// TIA Portal project "OCS_Portable_S300_To_S1500" (V14)

(* hardware
DEVICE "S7300/ET200M station_1"  S7-300 station
   slot 0: "Rail_0"  Rail  6ES7 390-1***0-0AA0
   slot 2: "PLC_1"  CPU 317-2 PN/DP  6ES7 317-2EK14-0AB0  V3.2
      slot 2: "PROFINET interface_1"  PN-IO
         slot 1: "Port_1"  Port
         slot 2: "Port_2"  Port
DEVICE "ET 200SP station_1"  ET 200SP-Station
   slot 0: "Rack_0"  Rack  6ES5 710-8MAx1
   slot 1: "PLC_2"  CPU 1512SP-1 PN  6ES7 512-1DK01-0AB0  V2.1
   slot 2: "TM Count 1x24V_1"  TM Count 1x24V  6ES7 138-6AA00-0BA0  V1.2
      slot 1: "TM Count 1x24V_1"  TM Count 1x24V
   slot 3: "CM PtP_1"  CM PtP  6ES7 137-6AA00-0BA0  V1.0
      slot 1: "CM PtP_1"  CM PtP Sub
   slot 4: "TM Pulse 2x24V_1"  TM Pulse 2x24V  6ES7 138-6DB00-0BB1  V1.0
      slot 1: "TM Pulse 2x24V_1"  TM Pulse 2x24V
   slot 5: "Server module_1"  Server module  6ES7 193-6PA00-0AA0  V1.1
      slot 1: "Server module_1"  Server module
   slot 127: "BA 2xRJ45"  BA 2xRJ45  6ES7 193-6AR00-0AA0  V0.0
      slot 32769: "Port_1"  6ES7 193-6AR00-0AA0
      slot 32770: "Port_2"  6ES7 193-6AR00-0AA0
*)

// ===== PLC "PLC_1"  CPU 317-2 PN/DP =====

VAR_GLOBAL   // PLC tag table "Merkers"
   "OSC_Work" AT %M20.5 : Bool;
END_VAR

DATA_BLOCK "Temp"   // DB1
{ S7_Optimized_Access := 'FALSE' }
VERSION : 0.1
   VAR
      Radians : Real;
   END_VAR
BEGIN
END_DATA_BLOCK

DATA_BLOCK "SU"   // DB101
{ S7_Optimized_Access := 'FALSE' }
VERSION : 0.1
   VAR
      su_Uac_6kV : Real;   // Действующее линейное напряжение AC на входе ЯВВ, В
      Spare_4_0 : Int;   // Резерв
      su_Fan_MD_QF1 : Bool;   // Автомат вентиляторов QF1 (0-выкл,1-вкл)
      su_Fan_MD_QF2 : Bool;   // Автомат вентиляторов QF2 (0-выкл,1-вкл)
      su_Fan_MD_QF3 : Bool;   // Автомат вентиляторов QF3 (0-выкл,1-вкл)
      su_Fan_MD_QF4 : Bool;   // Автомат вентиляторов QF4 (0-выкл,1-вкл)
      su_Fan_M1_ON : Bool;   // Контактор вентилятора КМ1 (0-выкл,1-вкл)
      su_Fan_M2_ON : Bool;   // Контактор вентилятора КМ2 (0-выкл,1-вкл)
      su_Fan_M6_ON : Bool;   // Контактор вентилятора КМ6 (0-выкл,1-вкл)
      su_Fan_M7_ON : Bool;   // Контактор вентилятора КМ7 (0-выкл,1-вкл)
      su_Fan_M8_ON : Bool;   // Контактор вентилятора КМ8 (0-выкл,1-вкл)
      su_Temp_ok : Bool;   // Температура в норме (0-выкл,1-вкл)
      su_Fan_MD_Ready : Bool;   // Готовность вентиляции ГП (0-выкл,1-вкл)
      su_Fan_M3_ON : Bool;   // Контактор вентилятора КМ3 (0-выкл,1-вкл)
      su_Fan_M4_ON : Bool;   // Контактор вентилятора КМ4 (0-выкл,1-вкл)
      su_Fan_M5_ON : Bool;   // Контактор вентилятора КМ5 (0-выкл,1-вкл)
      su_LH : Real;   // Длина подъемного каната, м
      su_LC : Real;   // Длина выдвижения рукояти, м
      su_OHRVD_AF : Bool;   // Ограничение хода рукояти. При выдвижении (0-ограничение выкл,1-ограничение)
      su_OHRVT_AF : Bool;   // Ограничение хода рукояти. При втягивании (0-ограничение выкл,1-ограничение)
      su_LC_Reset : Bool;   // Обнулить знчение энкодера напора (1-обнулить)
      su_OPK_AF : Bool;   // Ограничение подъема ковша (0-ограничение выкл, 1-ограничение)
      su_LH_Reset : Bool;   // Обнулить знчение энкодера подъема (1-обнулить)
      su_Field_Reduction : Bool;   // Ослабление поля (0-выкл,1-вкл)
      su_Field_Forcing : Bool;   // Форсировка поля (0-выкл,1-вкл)
      su_Autobrake_ON : Bool;   // Подхват тормозов (0-выкл,1-вкл)
      su_Brake_H : Bool;   // Тормоза привода подъема (1–расторможен,0–заторможен)
      su_Brake_C : Bool;   // Тормоза привода напора (1–расторможен,0–заторможен)
      su_Brake_S : Bool;   // Тормоза привода поворота (1–расторможен,0–заторможен)
      su_Brake_P : Bool;   // Тормоза привода хода левого (1–расторможен,0–заторможен)
      su_Brake_P_R : Bool;   // Тормоза привода хода правого (1–расторможен,0–заторможен)
      su_All_Protect : Bool;   // Автоматические защиты (0-выкл,1–вкл)
      su_BOS_Connect : Bool;   // Связь с БОС (0-связь есть,1-связи нет)
      su_Job_Limit : Bool;   // Уровень ограничения задания (0-задание 100%,1-задание 70%)
      su_Blocking_1 : Bool;   // Блокировка 1 Защита выше напорного вала (1-вкл,0-выкл)
      su_Blocking_2 : Bool;   // Блокировка 2 Защита при збросе ковша (1-вкл,0-выкл)
      su_Blocking_3 : Bool;   // Блокировка 3 Ограничение хода рукояти (1-вкл,0-выкл)
      su_Blocking_4 : Bool;   // Блокировка 4 Ограничение подъема ковша (1-вкл,0-выкл)
      su_Blocking_5 : Bool;   // Блокировка 5 Ограничение боковых нагрузок при черпании(1-вкл,0-выкл)
      su_Blocking_6 : Bool;   // Блокировка 6 Ограничение боковых нагрузок при работе с негабаритами(1-вкл,0-вык
      su_Blocking_7 : Bool;   // Блокировка 7 Передняя кромка(1-вкл,0-выкл)
      su_Blocking_8 : Bool;   // Блокировка 8 Защита от заброса стрелы(1-вкл,0-выкл)
      su_Blocking_9 : Bool;   // Блокировка 9 Ограничение длины разматывания подъемного каната (1-вкл,0-выкл)
      su_Enc_C_Connect : Bool;   // Энкодер напора подключен (1-связь есть,0-связи нет)
      su_Enc_H_Connect : Bool;   // Энкодер подъема подключен (1-связь есть,0-связи нет)
      Spare_19_3 : Bool;   // Резерв
      Spare_19_4 : Bool;   // Резерв
      Spare_19_5 : Bool;   // Резерв
      Spare_19_6 : Bool;   // Резерв
      Spare_19_7 : Bool;   // Резерв
      su_Job_H : DInt := DINT#0;   // Задание для привода подъема
      su_Job_S : DInt := DINT#0;   // Задание для привода поворота
      Spare_28_0 : Int;   // Резерв
      su_Excav : Bool;   // Режим "Экскавация" (1-вкл,0-выкл)
      su_Prop : Bool;   // Режим "Ход" (1-вкл,0-выкл)
      su_Work_S : Bool;   // Привод поворота расторможен (1-вкл,0-выкл)
      su_Work_C : Bool;   // Привод напора расторможен (1-вкл,0-выкл)
      su_Work_H : Bool;   // Привод подъема расторможен (1-вкл,0-выкл)
      su_Ready_S : Bool;   // Разрешение растормозить привод поворота (1-вкл,0-выкл)
      su_Fan_Prop : Bool;   // Вентиляторы двигателей хода (1-вкл,0-выкл)
      su_AR_Mode_Work : Bool;   // Активные выпрямители в режиме "Работа" (1-вкл,0-выкл)
      su_Ctrl_Is : Bool;   // Контроль изоляции (1-вкл,0-выкл)
      su_Ctrl_Ladder : Bool;   // Контроль положения лестницы (1-вкл,0-выкл)
      su_Relay_Alarm_ON : Bool;   // Реле включения аварии (1-вкл,0-выкл)
      su_Relay_CtrlC : Bool;   // Реле включения цепей управления (1-вкл,0-выкл)
      su_Ctrl_Breaker : Bool;   // Контроль состояния вводных автоматов (1-вкл,0-выкл)
      su_Limit_Switch : Bool;   // Конечные выключатели шкафов управления (1-вкл,0-выкл)
      su_Ready_P : Bool;   // Разрешение растормозить привод хода (1-вкл,0-выкл)
      su_Fan_Mot : Bool;   // Вентиляция машин (1-вкл,0-выкл)
      su_Work_P : Bool;   // Привод хода расторможен (1-вкл,0-выкл)
      su_Lubr : Bool;   // Смазка редукторов поворота (1-вкл,0-выкл)
      su_BUP_StartUp_ARm : Bool;   // Блок управления в режиме инициализации (1-вкл,0-выкл)
      su_BUP_ON_ARm : Bool;   // Блок управления в работе, управляющие импульсы поданы (1-вкл,0-выкл)
      su_BUP_StartUp_ARs1 : Bool;   // Блок управления в режиме инициализации (1-вкл,0-выкл)
      su_BUP_ON_ARs1 : Bool;   // Блок управления в работе, управляющие импульсы поданы (1-вкл,0-выкл)
      su_BUP_StartUp_ARs2 : Bool;   // Блок управления в режиме инициализации (1-вкл,0-выкл)
      su_BUP_ON_ARs2 : Bool;   // Блок управления в работе, управляющие импульсы поданы (1-вкл,0-выкл)
      su_BUP_StartUp_ARs3 : Bool;   // Блок управления в режиме инициализации (1-вкл,0-выкл)
      su_BUP_ON_ARs3 : Bool;   // Блок управления в работе, управляющие импульсы поданы (1-вкл,0-выкл)
      su_Magnet_M1H : Bool;   // Двигатель намагничен (1-вкл,0-выкл)
      su_BUP_StartUp_Hm : Bool;   // Блок управления в режиме инициализации (1-вкл,0-выкл)
      su_BUP_ON_Hm : Bool;   // Блок управления в работе, управляющие импульсы поданы (1-вкл,0-выкл)
      su_Magnet_M2H : Bool;   // Двигатель намагничен (1-вкл,0-выкл)
      su_BUP_StartUp_Hs : Bool;   // Блок управления в режиме инициализации (1-вкл,0-выкл)
      su_BUP_ON_Hs : Bool;   // Блок управления в работе, управляющие импульсы поданы (1-вкл,0-выкл)
      su_Magnet_MC : Bool;   // Двигатель намагничен (1-вкл,0-выкл)
      su_BUP_StartUp_C : Bool;   // Блок управления в режиме инициализации (1-вкл,0-выкл)
      su_BUP_ON_C : Bool;   // Блок управления в работе, управляющие импульсы поданы (1-вкл,0-выкл)
      su_Magnet_M1S : Bool;   // Двигатель намагничен (1-вкл,0-выкл)
      su_BUP_StartUp_Sm : Bool;   // Блок управления в режиме инициализации (1-вкл,0-выкл)
      su_BUP_ON_Sm : Bool;   // Блок управления в работе, управляющие импульсы поданы (1-вкл,0-выкл)
      su_Magnet_M2S : Bool;   // Двигатель намагничен (1-вкл,0-выкл)
      su_BUP_StartUp_Ss1 : Bool;   // Блок управления в режиме инициализации (1-вкл,0-выкл)
      su_BUP_ON_Ss1 : Bool;   // Блок управления в работе, управляющие импульсы поданы (1-вкл,0-выкл)
      su_Magnet_M3S : Bool;   // Двигатель намагничен (1-вкл,0-выкл)
      su_BUP_StartUp_Ss2 : Bool;   // Блок управления в режиме инициализации (1-вкл,0-выкл)
      su_BUP_ON_Ss2 : Bool;   // Блок управления в работе, управляющие импульсы поданы (1-вкл,0-выкл)
      su_Magnet_M4S : Bool;   // Двигатель намагничен (1-вкл,0-выкл)
      su_BUP_StartUp_Ss3 : Bool;   // Блок управления в режиме инициализации (1-вкл,0-выкл)
      su_BUP_ON_Ss3 : Bool;   // Блок управления в работе, управляющие импульсы поданы (1-вкл,0-выкл)
      su_Magnet_M1P : Bool;   // Двигатель намагничен (1-вкл,0-выкл)
      su_BUP_StartUp_C_P : Bool;   // Блок управления в режиме инициализации (1-вкл,0-выкл)
      su_BUP_ON_C_P : Bool;   // Блок управления в работе, управляющие импульсы поданы (1-вкл,0-выкл)
      su_Magnet_M2P : Bool;   // Двигатель намагничен (1-вкл,0-выкл)
      su_BUP_StartUp_S_P : Bool;   // Блок управления в режиме инициализации (1-вкл,0-выкл)
      su_BUP_ON_S_P : Bool;   // Блок управления в работе, управляющие импульсы поданы (1-вкл,0-выкл)
      Spare_36_5 : Bool;   // Резерв
      Spare_36_6 : Bool;   // Резерв
      Spare_36_7 : Bool;   // Резерв
      Spare_37_B : Byte;   // Резерв
      su_I_ARm : Real;   // Действующий ток, А
      su_Ud_ARm : Real;   // Напряжение звена постоянного тока, В
      su_Ia_ARm : Real;   // Амплитудный активный ток выпрямителя, А
      su_Ir_ARm : Real;   // Амплитудный индуктивный ток выпрямителя, А
      su_fs_ARm : Real;   // Частота сети
      su_Us_ARm : Real;   // Амплитудное напряжение на входе выпрямителя
      su_Pa_ARm : Real;   // Активная мощность выпрямителя
      su_I_ARs1 : Real;   // Действующий ток, А
      su_Ud_ARs1 : Real;   // Напряжение звена постоянного тока, В
      su_Ia_ARs1 : Real;   // Амплитудный активный ток выпрямителя, А
      su_Ir_ARs1 : Real;   // Амплитудный индуктивный ток выпрямителя, А
      su_fs_ARs1 : Real;   // Частота сети
      su_Us_ARs1 : Real;   // Амплитудное напряжение на входе выпрямителя
      su_Pa_ARs1 : Real;   // Активная мощность выпрямителя
      su_Job_I_ARs1 : Real;   // Задание на регулятор тока ведомого выпрямителя
      su_I_ARs2 : Real;   // Действующий ток, А
      su_Ud_ARs2 : Real;   // Напряжение звена постоянного тока, В
      su_Ia_ARs2 : Real;   // Амплитудный активный ток выпрямителя, А
      su_Ir_ARs2 : Real;   // Амплитудный индуктивный ток выпрямителя, А
      su_fs_ARs2 : Real;   // Частота сети
      su_Us_ARs2 : Real;   // Амплитудное напряжение на входе выпрямителя
      su_Pa_ARs2 : Real;   // Активная мощность выпрямителя
      su_Job_I_ARs2 : Real;   // Задание на регулятор тока ведомого выпрямителя
      su_I_ARs3 : Real;   // Действующий ток, А
      su_Ud_ARs3 : Real;   // Напряжение звена постоянного тока, В
      su_Ia_ARs3 : Real;   // Амплитудный активный ток выпрямителя, А
      su_Ir_ARs3 : Real;   // Амплитудный индуктивный ток выпрямителя, А
      su_fs_ARs3 : Real;   // Частота сети
      su_Us_ARs3 : Real;   // Амплитудное напряжение на входе выпрямителя
      su_Pa_ARs3 : Real;   // Активная мощность выпрямителя
      su_Job_I_ARs3 : Real;   // Задание на регулятор тока ведомого выпрямителя
      su_I_M1H : Real;   // Действующий ток статора, А
      su_Ud_Hm : Real;   // Напряжение звена постоянного тока, В
      su_Id_M1H : Real;   // Ток намагничивания статора, А
      su_Iq_M1H : Real;   // Активный ток статора, А
      su_W_M1H : Real;   // Скорость, рад/с
      su_Psi2_M1H : Real;   // Поток ротора, Вб
      su_U_M1H : Real;   // Фазное напряжение двигателя, В
      su_JobW_Hm : Real;   // Задание на скорость, ед
      su_I_M2H : Real;   // Действующий ток статора, А
      su_Ud_Hs : Real;   // Напряжение звена постоянного тока, В
      su_Id_M2H : Real;   // Ток намагничивания статора, А
      su_Iq_M2H : Real;   // Активный ток статора, А
      su_W_M2H : Real;   // Скорость, рад/с
      su_Psi2_M2H : Real;   // Поток ротора, Вб
      su_U_M2H : Real;   // Фазное напряжение двигателя, В
      su_JobW_Hs : Real;   // Задание на скорость, ед
      su_I_MC : Real;   // Действующий ток статора, А
      su_Ud_C : Real;   // Напряжение звена постоянного тока, В
      su_Id_MC : Real;   // Ток намагничивания статора, А
      su_Iq_MC : Real;   // Активный ток статора, А
      su_W_MC : Real;   // Скорость, рад/с
      su_Psi2_MC : Real;   // Поток ротора, Вб
      su_U_MC : Real;   // Фазное напряжение двигателя, В
      su_JobW_C : Real;   // Задание на скорость, ед
      su_I_M1S : Real;   // Действующий ток статора, А
      su_Ud_Sm : Real;   // Напряжение звена постоянного тока, В
      su_Id_M1S : Real;   // Ток намагничивания статора, А
      su_Iq_M1S : Real;   // Активный ток статора, А
      su_W_M1S : Real;   // Скорость, рад/с
      su_Psi2_M1S : Real;   // Поток ротора, Вб
      su_U_M1S : Real;   // Фазное напряжение двигателя, В
      su_JobW_Sm : Real;   // Задание на скорость, ед
      su_I_M2S : Real;   // Действующий ток статора, А
      su_Ud_Ss1 : Real;   // Напряжение звена постоянного тока, В
      su_Id_M2S : Real;   // Ток намагничивания статора, А
      su_Iq_M2S : Real;   // Активный ток статора, А
      su_W_M2S : Real;   // Скорость, рад/с
      su_Psi2_M2S : Real;   // Поток ротора, Вб
      su_U_M2S : Real;   // Фазное напряжение двигателя, В
      su_JobW_Ss1 : Real;   // Задание на скорость, ед
      Spare_322_0 : Real;   // Резерв
      su_State_H1 : Bool;   // Готовность преобразователя подъема 1 (0-авария,1-готов)
      su_State_H2 : Bool;   // Готовность преобразователя подъема 2 (0-авария,1-готов)
      su_State_C : Bool;   // Готовность преобразователя напора (0-авария,1-готов)
      su_State_P1 : Bool;   // Готовность преобразователя хода 1 (0-авария,1-готов)
      su_State_P2 : Bool;   // Готовность преобразователя хода 2 (0-авария,1-готов)
      su_State_S1 : Bool;   // Готовность преобразователя поворота 1 (0-авария,1-готов)
      su_Overheat_TS : Bool;   // Перегрев силового трансформатора (0-авария,1-готов)
      su_GB_Charge : Bool;   // Блок заряда аккумуляторов (0-авария,1-готов)
      su_Relay_K4 : Bool;   // Реле К4 резерв (0-выкл,1-вкл)
      su_Relay_K3 : Bool;   // Реле К3, готовность блоков сброса (0-выкл,1-вкл)
      su_Relay_K2 : Bool;   // Реле К2 включение ВВ контактора (0-выкл,1-вкл)
      su_State_AR1 : Bool;   // Готовность активного выпрямителя 1 (0-авария,1-готов)
      su_State_AR2 : Bool;   // Готовность активного выпрямителя 2 (0-авария,1-готов)
      su_State_AR3 : Bool;   // Готовность активного выпрямителя 3 (0-авария,1-готов)
      su_State_Chop1 : Bool;   // Блок сброс 1 (0-авария,1-готов)
      su_State_Chop2 : Bool;   // Блок сброс 2 (0-авария,1-готов)
      su_Relay_K7 : Bool;   // Реле К7 резерв (0-выкл,1-вкл)
      su_Relay_K6 : Bool;   // Реле К6 резерв (0-выкл,1-вкл)
      su_State_AR4 : Bool;   // Готовность активного выпрямителя 4 (0-авария,1-готов)
      su_Relay_K5 : Bool;   // Реле К5 резерв (0-выкл,1-вкл)
      su_Relay_K1 : Bool;   // Реле К1 включение готовности преобразователей ГП (0-выкл,1-вкл)
      su_Vent_MD : Bool;   // Вентиляция главных приводов (0-выкл,1-вкл)
      su_HV_Contactor_ON : Bool;   // ВВ контактор включен (0-выкл,1-вкл)
      su_State_S2 : Bool;   // Готовность преобразователя поворота 2 (0-авария,1-готов)
      su_State_S3 : Bool;   // Готовность преобразователя поворота 3 (0-авария,1-готов)
      su_State_S4 : Bool;   // Готовность преобразователя поворота 4 (0-авария,1-готов)
      Spare_329_2 : Bool;   // Резерв
      Spare_329_3 : Bool;   // Резерв
      Spare_329_4 : Bool;   // Резерв
      Spare_329_5 : Bool;   // Резерв
      Spare_329_6 : Bool;   // Резерв
      Spare_329_7 : Bool;   // Резерв
      su_BOS_Enc_H : Int;   // Значение БОСЭ механизма подъема (1 оборот 2^10 бит)
      su_BOS_Enc_C : Int;   // Значение БОСЭ механизма напора (1 оборот 2^10 бит)
      su_MD_OFF : Bool;   // Отключение главных приводов (0-выкл,1-вкл)
      su_VH : Real;   // Линейная скорость подъема
      su_VC : Real;   // Линейная скорость напора
      su_Job_C : DInt := DINT#0;   // Задание для привода напора
      su_Ia_PowerT : Real;   // Ток в фазе А первичной обмотки силового трансформатора, А
      su_Ib_PowerT : Real;   // Ток в фазе В первичной обмотки силового трансформатора, А
      su_I_M3S : Real;   // Действующий ток статора, А
      su_Ud_Ss2 : Real;   // Напряжение звена постоянного тока, В
      su_Id_M3S : Real;   // Ток намагничивания статора, А
      su_Iq_M3S : Real;   // Активный ток статора, А
      su_W_M3S : Real;   // Скорость, рад/с
      su_Psi2_M3S : Real;   // Поток ротора, Вб
      su_U_M3S : Real;   // Фазное напряжение двигателя, В
      su_JobW_Ss2 : Real;   // Задание на скорость, ед
      su_I_M4S : Real;   // Действующий ток статора, А
      su_Ud_Ss3 : Real;   // Напряжение звена постоянного тока, В
      su_Id_M4S : Real;   // Ток намагничивания статора, А
      su_Iq_M4S : Real;   // Активный ток статора, А
      su_W_M4S : Real;   // Скорость, рад/с
      su_Psi2_M4S : Real;   // Поток ротора, Вб
      su_U_M4S : Real;   // Фазное напряжение двигателя, В
      su_JobW_Ss3 : Real;   // Задание на скорость, ед
      su_I_M1P : Real;   // Действующий ток статора, А
      su_Ud_C_P : Real;   // Напряжение звена постоянного тока, В
      su_Id_M1P : Real;   // Ток намагничивания статора, А
      su_Iq_M1P : Real;   // Активный ток статора, А
      su_W_M1P : Real;   // Скорость, рад/с
      su_Psi2_M1P : Real;   // Поток ротора, Вб
      su_U_M1P : Real;   // Фазное напряжение двигателя, В
      su_JobW_C_P : Real;   // Задание на скорость, ед
      su_I_M2P : Real;   // Действующий ток статора, А
      su_Ud_S_P : Real;   // Напряжение звена постоянного тока, В
      su_Id_M2P : Real;   // Ток намагничивания статора, А
      su_Iq_M2P : Real;   // Активный ток статора, А
      su_W_M2P : Real;   // Скорость, рад/с
      su_Psi2_M2P : Real;   // Поток ротора, Вб
      su_U_M2P : Real;   // Фазное напряжение двигателя, В
      su_JobW_S_P : Real;   // Задание на скорость, ед
      su_BUARm_ID : Int;   // Номер блока активного выпрямителя ведущего
      su_BUARs1_ID : Int;   // Номер блока активного выпрямителя ведомого 1
      su_BUARs2_ID : Int;   // Номер блока активного выпрямителя ведомого 2
      su_BUARs3_ID : Int;   // Номер блока активного выпрямителя ведомого 3
      su_Type_AR : Int;   // Текущий тип преобразователя
      su_BUP_Hm_ID : Int;   // Номер БУПа привода подъема ведущего
      su_BUP_Hs_ID : Int;   // Номер БУПа привода подъема ведомого
      su_BUP_C_ID : Int;   // Номер БУПа привода напора
      su_BUP_Sm_ID : Int;   // Номер БУПа привода поворота ведущего
      su_BUP_Ss1_ID : Int;   // Номер БУПа привода поворота ведомого 1
      su_BUP_Ss2_ID : Int;   // Номер БУПа привода поворота ведомого 2
      su_BUP_Ss3_ID : Int;   // Номер БУПа привода поворота ведомого 3
      su_BUP_CP_ID : Int;   // Номер БУПа привода напора-хода
      su_BUP_SP_ID : Int;   // Номер БУПа привода поворота-хода
      su_Type_Pr : Int;   // Текущий тип привода
      su_Temp_ARm : Int;   // Средняя температура активного выпрямителя ведущего
      su_Temp_ARs1 : Int;   // Средняя температура активного выпрямителя ведомого 1
      su_Temp_ARs3 : Int;   // Средняя температура активного выпрямителя ведомого 2
      su_Temp_ARs2 : Int;   // Средняя температура активного выпрямителя ведомого 3
      su_Temp_Hm : Int;   // Средняя температура преобразователя подъема ведущего
      su_Wr_M1H : Int;   // Электрическая скорость ротора M1H (показания датчика, рад/с)
      su_Temp_Hs : Int;   // Средняя температура преобразователя подъема ведомого
      su_Wr_M2H : Int;   // Электрическая скорость ротора M2H (показания датчика, рад/с)
      su_Temp_C : Int;   // Средняя температура преобразователя напора
      su_Wr_MC : Int;   // Электрическая скорость ротора MC (показания датчика, рад/с)
      su_Temp_Sm : Int;   // Средняя температура преобразователя поворота ведущего
      su_Wr_M1S : Int;   // Электрическая скорость ротора M1S (показания датчика, рад/с)
      su_Temp_Ss1 : Int;   // Средняя температура преобразователя поворота ведомого 1
      su_Wr_M2S : Int;   // Электрическая скорость ротора M2S (показания датчика, рад/с)
      su_Temp_Ss2 : Int;   // Средняя температура преобразователя поворота ведомого 2
      su_Wr_M3S : Int;   // Электрическая скорость ротора M3S (показания датчика, рад/с)
      su_Temp_Ss3 : Int;   // Средняя температура преобразователя поворота ведомого 3
      su_Wr_M4S : Int;   // Электрическая скорость ротора M4S (показания датчика, рад/с)
      su_Temp_C_P : Int;   // Средняя температура преобразователя напора-хода
      su_Wr_M1P : Int;   // Электрическая скорость ротора M1P (показания датчика, рад/с)
      su_Temp_S_P : Int;   // Средняя температура преобразователя поворота-хода
      su_Wr_M2P : Int;   // Электрическая скорость ротора M2P (показания датчика, рад/с)
      su_I_M1H_fs : Real;   // Действующий ток статора, A (быстрое значение)
      su_Id_M1H_fs : Real;   // Ток намагничивания статора, А (быстрое значение)
      su_Iq_M1H_fs : Real := -0.375;   // Активный ток статора, А (быстрое значение)
      su_W_M1H_fs : Real;   // Скорость, рад/с (быстрое значение)
      su_I_C_fs : Real;   // Действующий ток статора, A (быстрое значение)
      su_Id_C_fs : Real;   // Ток намагничивания статора, А (быстрое значение)
      su_Iq_C_fs : Real;   // Активный ток статора, А (быстрое значение)
      su_W_C_fs : Real;   // Скорость, рад/с (быстрое значение)
      su_I_S_fs : Real;   // Действующий ток статора, A (быстрое значение)
      su_Id_S_fs : Real;   // Ток намагничивания статора, А (быстрое значение)
      su_Iq_S_fs : Real := 59.75;   // Активный ток статора, А (быстрое значение)
      su_W_S_fs : Real;   // Скорость, рад/с (быстрое значение)
   END_VAR
BEGIN
END_DATA_BLOCK

DATA_BLOCK "AP"   // DB103
{ S7_Optimized_Access := 'FALSE' }
VERSION : 0.1
   VAR
      ap_QF_FanMD_Off : Bool;   // отключен автомат вентиляторов главных приводов
      ap_UZ_FanMD_On : Bool;   // преобразователь пуска вентиляторов главных приводов включен
      ap_QF_FanProp_Off : Bool;   // отключен автомат вентиляторов двигателей хода
      ap_UZ_FanProp_On : Bool;   // преобразователь пуска вентиляторов двигателей хода включен
      ap_QF_KB_On : Bool;   // автомат преобразователя кабельного барабана включен
      ap_QF_ODK_On : Bool;   // автомат преобразователя открывания днища ковша включен
      ap_PS_110v_On : Bool;   // питание источника 110В включено
      ap_CtrlC_110v_On : Bool;   // питание цепей управления 110В включено
      ap_Gudok : Bool;   // пневмосигнал включен
      ap_ODK : Bool;   // управление УДК
      ap_Vent_Prop_On : Bool;   // вентиляция привода хода включена
      ap_Vent_MD_On : Bool;   // вентиляция главных приводов включена
      ap_QF_FVU12_On : Bool;   // общий автомат ФВУ включен
      ap_FVU12_On : Bool;   // ФВУ включены
      ap_QF_FVU1_On : Bool;   // автомат ФВУ1 включен
      ap_QF_FVU2_On : Bool;   // автомат ФВУ2 включен
      ap_QF_Fan_Kuzov : Bool;   // автомат вентилятора кузова включен
      ap_Vent_Kuzov : Bool;   // вентиляция кузова включена
      ap_FVU1_FVU2_On : Bool;   // ФВУ1 или(и) ФВУ2 включен
      ap_QF_Lubr : Bool;   // общий автомат смазки редукторов поворота включен(0)
      ap_Lubr_On : Bool;   // смазка редукторов поворота включена
      ap_QF_Heat : Bool;   // общий автомат нагревателей смазки редукторов поворота включен
      ap_Heat_M1S : Bool;   // нагреватели ЕК1-ЕК6 включены
      ap_Heat_M2S : Bool;   // нагреватели ЕК7-ЕК12 включены
      ap_Heat_M3S : Bool;   // нагреватели ЕК13-ЕК18 включены
      ap_Heat_M4S : Bool;   // нагреватели ЕК19-ЕК23 включены
      ap_QF_Komr : Bool;   // компрессорная установка включена
      ap_QF_ACSS380V : Bool;   // станция густой смазки включена
      ap_QF_Vvod380 : Bool;   // вводной автоматический выключатель 380В включен
      ap_QF_TV3 : Bool;   // выключатель трансформатора TV3 включен
      ap_QF_TV2M : Bool;   // выключатель трансформатора TV2M включен
      ap_QF_Vent_SHGP : Bool;   // выключатель вентиляции ШГП включен
      ap_QF_Light : Bool;   // выключатель прожекторного освещения включен
      ap_QF_CtrlC24V : Bool;   // выключатель цепей управления -24В включен
      ap_QF_YAVV220V : Bool;   // выключатель цепей управления ЯВВ(220В) включен
      ap_QF_Charge_ZPT : Bool;   // выключатель цепей заряда конденсаторов включен
      ap_QF_BKTT220V : Bool;   // выключатель блока контроля температуры(220В) включен
      ap_QF_IS220V : Bool;   // выключатель ИС (220В) включен
      ap_QF_ACSS220V : Bool;   // выключатель обогрева шкафа густой смазки включен
      ap_KM_TV3 : Bool;   // трансформатор освещения TV3 включен
      ap_KM_Light : Bool;   // прожекторное освещение включен
      ap_KM_Heat_H : Bool;   // Контактор обогревателей масла редуктора подъЁма
      ap_QF_Heat_H : Bool;   // Автомат обогревателей масла редуктора подъЁма
   END_VAR
BEGIN
END_DATA_BLOCK

DATA_BLOCK "BD"   // DB120
{ S7_Optimized_Access := 'FALSE' }
VERSION : 0.1
   VAR
      n_Brig : Int;   // Номер бригады
      wt_H_Hour : DInt := DINT#0;   // Часы работы механизма подъёма
      wt_H_Minut : Int;   // Минуты работы механизма подъёма
      wt_H_Second : Int;   // Секунды работы механизма подъёма
      wt_C_Hour : DInt := DINT#0;   // Часы работы механизма напора
      wt_C_Minut : Int;   // Минуты работы механизма напора
      wt_C_Second : Int;   // Секунды работы механизма напора
      wt_S_Hour : DInt := DINT#0;   // Часы работы механизма поворота
      wt_S_Minut : Int;   // Минуты работы механизма поворота
      wt_S_Second : Int;   // Секунды работы механизма поворота
      wt_P_Hour : DInt := DINT#0;   // Часы работы механизма хода
      wt_P_Minut : Int;   // Минуты работы механизма хода
      wt_P_Second : Int;   // Секунды работы механизма хода
      wt_Exc_Hour : DInt := DINT#0;   // Время основной работы (Час)
      wt_Exc_Min : Int;   // Время основной работы (Минут)
      wt_Exc_Sec : Int;   // Время основной работы (Секунд)
      odo_Prop_all : Real;   // Общий пробег за время эксплуатации
      Spare_I_1 : Int;   // Резерв
      Spare_I_2 : Int;   // Резерв
      wt_Prop_Hour : DInt := DINT#0;   // Время хода (Час)
      wt_Prop_Min : Int;   // Время хода (Минут)
      wt_Prop_Sec : Int;   // Время хода (Секунд)
      wt_Idle_Hour : DInt := DINT#0;   // Время простоя (Час)
      wt_Idle_Min : Int;   // Время простоя (Минут)
      wt_Idle_Sec : Int;   // Время простоя (Секунд)
      wt_UG_Hour : DInt := DINT#0;   // Время работы при косом стоянии (Час)
      wt_UG_Min : Int;   // Время работы при косом стоянии (Минут)
      wt_UG_Sec : Int;   // Время работы при косом стоянии (Секунд)
      Mas_Basket : Real;   // Масса грунта в ковше (кг)
      Mas_TS_cr : Real;   // Масса грунта в ТС текущая (кг)
      Mas_TS_lst : Real;   // Масса грунта в последнем ТС (кг)
      Mas_TS_all : Real;   // Масса грунта общая (кг)
      AE1_st : Real;   // Активная потреблённая энергия в начале смены
      AE2_st : Real;   // Активная отданная энергия в начале смены
      RE1_st : Real;   // Реактивная потреблённая энергия в начале смены
      RE2_st : Real;   // Реактивная отданная энергия в начале смены
      AE1_cr : Real;   // Активная потреблённая энергия за смену
      AE2_cr : Real;   // Активная отданная энергия за смену
      RE1_cr : Real;   // Реактивная потреблённая энергия за смену
      RE2_cr : Real;   // Реактивная отданная энергия за смену
      AE1_all : Real;   // Активная потреблённая энергия общая
      AE2_all : Real;   // Активная отданная энергия общая
      RE1_all : Real;   // Реактивная потреблённая энергия общая
      RE2_all : Real;   // Реактивная отданная энергия общая
      tm_Reg_H : Int;   // Время регистрации бригады (час)
      tm_Reg_M : Int;   // Время регистрации бригады (мин)
      n_TS : Int;   // Количество погруженных ТС
      TS_Num : Int;   // Грузоподъёмность текущего ТС
      TS_1 : Int;   // Грузоподъёмность трансп.ср-ва 1
      TS_2 : Int;   // Грузоподъёмность трансп.ср-ва 2
      TS_3 : Int;   // Грузоподъёмность трансп.ср-ва 3
      TS_4 : Int;   // Грузоподъёмность трансп.ср-ва 4
      sm_Duration : Int;   // Продолжительность смены
      sm_Hour : Int;   // Начало первой смены. Час.
      sm_Min : Int;   // Начало первой смены. Мин.
      Shft_Reg : Bool;   // Флаг регистрации бригады
      fl_Pogr_On : Bool;   // Флаг погрузки
      Spare_160_2 : Bool;   // Резерв
      Spare_160_3 : Bool;   // Резерв
      Spare_160_4 : Bool;   // Резерв
      Spare_160_5 : Bool;   // Резерв
      Spare_160_6 : Bool;   // Резерв
      Spare_160_7 : Bool;   // Резерв
      tm_Reg_Mnt : Int;   // Время регистрации бригады (месяц)
      tm_Reg_Day : Int;   // Время регистрации бригады (год)
      kVAh_Total : DInt := DINT#0;   // Общая полная мощность
      Frequency : Real;   // Частота сети
      U_12 : Int;   // Напряжение между фазами 1 и 2
      U_23 : Int;   // Напряжение между фазами 2 и 3
      U_31 : Int;   // Напряжение между фазами 3 и 1
      PASS : Word;   // Эти три заглушки тут нужны чтобы адреса не съехали
      PASS1 : Word;   // Эти три заглушки тут нужны чтобы адреса не съехали
      PASS2 : Word;   // Эти три заглушки тут нужны чтобы адреса не съехали
      I_1 : Real;   // Ток фазы 1
      I_2 : Real;   // Ток фазы 2
      I_3 : Real;   // Ток фазы 3
      PF : Real;   // Сдвиг фаз
      Count_BTL_ErrPoint_2 : Int;   // Количество забросов за вторую точку
   END_VAR
BEGIN
END_DATA_BLOCK

DATA_BLOCK "Work"   // DB121
TITLE = Данные для работы
{ S7_Optimized_Access := 'FALSE' }
VERSION : 0.1
   VAR
      on_SU : Bool;   // Система управления в работе
      pH_On : Bool;   // Привод подьёма включен
      pS_On : Bool;   // Привод поворота включен
      pC_On : Bool;   // Привод напора включен
      pP_On : Bool;   // Привод хода включен
      p_On : Bool;   // Главные приводы включены
      ACSS_On : Bool;   // АЦСС в работе
      HMI_On : Bool;   // HMI в работе
      Auto_Park : Bool;   // Команда на автоматическую парковку компьютера
      Ack_Alrm : Bool;   // Квитирование алармов
      T_Set_on : Bool;   // Команда на установку времени
      fl_Reset_LH : Bool;   // Флаг сброса длины каната подъёма
      fl_Reset_LC : Bool;   // Флаг сброса длины рукояти
      on_Auto_Def : Bool;   // Включение / отключение автозащит
      Reset_flt_SU : Bool;   // Сброс ошибок системы управления
      LK_ON : Bool;   // Вывод левой камеры
      cnt_Sec : Int;   // Счётчик секунд
      ABS_U : Int;   // Абсолютный угол поворота
      Spare_w6 : Word;   // Уставка паузы P1
      ug_Prod_Mx : Real;   // Угол наклона экскаватора продольная плоскость предыдущий
      ug_Popr_Mx : Real;   // Угол наклона экскаватора поперечная плоскость предыдущий
      ug_Prod_Mn : Real;   // Разность между тек. и пред. уголаами в продольной плоскости
      ug_Popr_Mn : Real;   // Разность между тек. и пред. уголаами в поперечной плоскости
      ug_Prod_MAX : Real;   // Разность между тек. и пред. уголаами в продольной плоскости макс.
      ug_Popr_MAX : Real;   // Разность между тек. и пред. уголаами в поперечной плоскости макс.
      ABS_H : Real;   // Абсолютная скорость подъёма
      Spare_I36 : Int;   // Счётчик лайфбитов АЦСС
      Spare_I38 : Int;   // Предыдущий лайфбит АЦСС
      HMI_LB : Int;   // Лайфбит HMI
      HMI_LB_Cnt : Int;   // Счётчик лайфбитов HMI
      HMI_LB_Pred : Int;   // Предыдущий лайфбит HMI
      smf_ACSS : Int;   // Суммарный фолт системы смазки
      smf_Tmpr : Int;   // Суммарный фолт температур
      Act_Time_Year : Int;   // Текущая дата/время - Год
      Act_Time_Month : Int;   // Текущая дата/время - Месяц
      Act_Time_Day : Int;   // Текущая дата/время - День
      Act_Time_Hour : Int;   // Текущая дата/время - Час
      Act_Time_Min : Int;   // Текущая дата/время - Минуты
      Act_Time_Sec : Int;   // Текущая дата/время - Секунды
      smf_AP : Int;   // Суммарный фолт вспомогательных приводов
      smf_GP : Int;   // Суммарный фолт главных приводов
      fl_WC_Start : Bool;   // Флаг начала рабочего цикла
      Spare_66_1 : Bool;   // Резерв
      Spare_66_2 : Bool;   // Резерв
      Reg_Lim_BN : Bool;   // Режим ограничения по боковым нагрузкам
      fl_Blok_BN : Bool;   // Флаг блокировки защиты от боковых нагрузок
      fl_Kach : Bool;   // Флаг измерения качания
      fl_S_Final : Bool;   // Флаг завершения смены
      Spare_66_7 : Bool;   // Резерв
      fl_WC_Idle : Bool;   // Флаг простоя
      fl_WC_Drag : Bool;   // Флаг черпания
      fl_WC_S_Rz : Bool;   // Флаг поворота разгрузку
      fl_WC_Rz : Bool;   // Флаг разгрузи
      fl_WC_S_Zb : Bool;   // Флаг поворота в забой
      fl_WC_Prop : Bool;   // Флаг хода
      fl_WC_Wait : Bool;   // Флаг ожидания транспорта
      Spare_67_7 : Bool;   // Резерв
      Spare_W68 : Word;   // Резерв
      lim_VH : Byte;   // Ограничение скорости подъёма
      lim_VS : Byte;   // Ограничение скорости поворота
      lim_VC : Byte;   // Ограничение скорости напора
      lim_IsH : Byte;   // Ограничение стопорного тока подъёма
      lim_IsS : Byte;   // Ограничение стопорного тока поворота
      lim_IsC : Byte;   // Ограничение стопорного тока напора
      ug_Pov_Tk : Int;   // Угол поворота платформы экскаватора текущий
      cmd_SU : Byte;   // Команда системе управления
      cnt_Zub : Int;   // Счётчик зубъев
      fl_Entg_Res : Bool;   // Флаг сброса счётчика
      Win_Protect : Bool;   // Флаг работы в зимнее время
      Shft_f_Reg : Bool;   // Флаг первой регистрации бригады
      fl_Excs : Bool;   // Флаг экскавации
      fl_Prop : Bool;   // Флаг перемещения
      fl_Idle : Bool;   // Флаг простоя
      Camera_ON : Bool;   // Включение камеры
      Camera_FIN : Bool;   // Отключение камеры
      fl_Second : Bool;   // Фронт секунд
      Reg_Lim_Turn : Bool;   // Режим ограничений от недопустимого разворота
      Reset_Enrg : Bool;   // Сброс счётчика
      fl_KS : Bool;   // Флаг работы при косом стоянии
      Winter_Pr_Removing : Bool;   // Процесс снятия зимних защит запущен
      ACSS_Starting_Now : Bool;   // Выполняется запуск системы смазки (0-нет; 1-да)
      ACSS_SumBypass : Bool;   // Суммарный байпасс питателей системы смазки
      RB_HMI : Bool;   // Эмулятор правой кнопки командоаппарата с HMI
      Camera_Reg : Int;   // Режим работы камеры
      smf_Komp : Int;   // Суммарный фолт компрессора
      ABS_Sw : Real;   // Абсолютная скорость поворота
      Reg_WC : Int;   // Режим рабочего цикла (1-черпание,2-пов.на разгр,3-разгр,4-поворот в заб.)
      ug_Povorota : Int;   // Угол поворота платформы экскаватора
      Prc_TS : Int;   // Процент заполнения самосвала
      dp_ET_2 : Bool;   // Флаг работы станции ET200 в шкафу АИС2
      dp_ET_3 : Bool;   // Флаг работы станции ET200 в шкафу АИС3
      dp_ET_4 : Bool;   // Флаг работы станции ET200 в шкафу АИС4
      dp_ACSS : Bool;   // Флаг работы контроллера густой смазки
      dp_CAN_AP : Bool;   // Флаг работы шлюза CAN-DP вспом. приводов
      dp_CAN_GP : Bool;   // Флаг работы шлюза CAN-DP гл. приводов
      dp_GNAMG : Bool;   // Флаг работы инклинометра
      dp_KOMPR : Bool;   // Флаг работы компрессора
      fl_Wint_Pr : Bool;   // Флаг защиты МК при работе зимой
      fl_Win_Pr_St_Res : Bool;   // Флаг старта процедуры сброса
      Reg_Lim_UG : Bool;   // Режим ограничения по углу стояния
      Reg_Lim_ZS : Bool;   // Режим ограничения от заброса стрелы
      Reg_Lim_Winter : Bool;   // Режим ограничения зимой
      Reg_Lim_HMI : Bool;   // Режим ограничения с HMI
      bl_Rdy : Bool;   // Флаг готовности БУП к обработке сообщений
      bl_A_Rdy : Bool;   // Флаг готовности БУАВ к обработке сообщений
      DT_Wint_Res : Date_And_Time;   // Дата и время отключения защит в зимнее время
      lb_PLC : Int;   // Лайфбит PLC
      smf_ACSS_A1 : Int;   // Суммарный фолт станции A1 системы смазки
      smf_ACSS_A2 : Int;   // Суммарный фолт станции A2 системы смазки
      smf_ACSS_H1 : Int;   // Суммарный фолт станции H1 системы смазки
      tm_WP_Reset : DInt := DINT#0;   // Время до снятия зимних защит mc
      Offset : Int;   // Сдвиг в блоке данных старых алармов
      lim_VH_HMI : Byte;   // Ограничение скорости подъёма с HMI
      lim_VS_HMI : Byte;   // Ограничение скорости поворота с HMI
      lim_VC_HMI : Byte;   // Ограничение скорости напора с HMI
      lim_IsH_HMI : Byte;   // Ограничение стопорного тока подъёма с HMI
      lim_IsS_HMI : Byte;   // Ограничение стопорного тока поворота с HMI
      lim_IsC_HMI : Byte;   // Ограничение стопорного тока напора с HMI
      n_BUP_cr : Int;   // Текущий номер БУП
      n_BUP_pr : Int;   // Предыдущий номер БУП
      cnt_BUP : Int;   // Счётчик БУП
      n_BUP : Array[1..15] of Int;   // Массив номеров блоков
      t_BUP : Array[1..15] of Int;   // Массив типов блоков
      SU_LB : Int;   // Лайфбит СУ
      SU_LB_Cnt : Int;   // Счётчик лайфбитов СУ
      SU_LB_Pred : Int;   // Предыдущий лайфбит СУ
      QwrSATEC : DWord;   // Формируемое двойное слово запроса, отправляемое в счётчик электроэнергии
      PASS_SATEC : DWord := DWORD#16#0101_0E14;   // Заготовка для посылки: byte0(0001 0100)byte1(0000 1110)ID-0x0101
      Control_Run_FC114 : Int;   // Здесь лежит байт, управляющий чтением показаний с SADEC
      su_LH_prev : Real;   // Предыдущая (50Гц) длина подъемного каната м
      su_LC_prev : Real;   // Предыдущая (50Гц) длина выдвижения рукояти м
      V_prop_left : Real;   // Скорость движения левой гусеницы
      V_prop_right : Real;   // Скорость движения правой гусеницы
      su_W_M1P_Pred : Real;   // Скорость двигателя хода M1P в предыдущем скане
      su_W_M2P_Pred : Real;   // Скорость двигателя хода M2P в предыдущем скане
      W_pP_Pred : Real;   // Cредняя скорость привода хода в предыдущем скане
      W_pP_Cr : Real;   // Cредняя скорость привода хода в текущем скане
      ABS_W_pP_Pred : Real;   // Абсолютное значение средней скорости привода хода в предыдущем скане
      ABS_W_pP_Cr : Real;   // Абсолютное значение средней скорости привода хода в текущем скане
      odo_Prop_cr : Real;   // Пробег за один шаг интегрирования
      lim_VP_M1P : Byte;   // Ограничение скорости левой гусеницы
      lim_VP_M2p : Byte;   // Ограничение скорости правой гусеницы
   END_VAR
BEGIN
END_DATA_BLOCK

DATA_BLOCK "DB_OSC"   // DB505
{ S7_Optimized_Access := 'FALSE' }
VERSION : 0.1
   VAR
      Act : Int;   // Флаг работы осцилографа
      Ready : Int;   // Флаг готовности массивов к передаче
      Cnt : Int;   // Счётчик параметров
      Ramp : Int;   // Пила
      Max_Addr : DInt := DINT#0;   // Максимальный адрес текущего массива
      cr_Addr_1 : DInt := DINT#0;   // Текущий адрес массива канала 1
      cr_Addr_2 : DInt := DINT#0;   // Текущий адрес массива канала 2
      cr_Addr_3 : DInt := DINT#0;   // Текущий адрес массива канала 3
      cr_Addr_4 : DInt := DINT#0;   // Текущий адрес массива канала 4
      cr_Addr_5 : DInt := DINT#0;   // Текущий адрес массива канала 5
      cr_Addr_6 : DInt := DINT#0;   // Текущий адрес массива канала 6
      cr_Addr_7 : DInt := DINT#0;   // Текущий адрес массива канала 7
      cr_Addr_8 : DInt := DINT#0;   // Текущий адрес массива канала 8
      cr_Addr_9 : DInt := DINT#0;   // Текущий адрес массива канала 9
      cr_Addr_10 : DInt := DINT#0;   // Текущий адрес массива канала 10
      cr_Addr_Rmp : DInt := DINT#32448;   // Текущий адрес пилы
      ar_Ch_01 : Array[1..200] of Int;   // Массив значений канала 1
      ar_Ch_02 : Array[1..200] of Int;   // Массив значений канала 2
      ar_Ch_03 : Array[1..200] of Int;   // Массив значений канала 3
      ar_Ch_04 : Array[1..200] of Int;   // Массив значений канала 4
      ar_Ch_05 : Array[1..200] of Int;   // Массив значений канала 5
      ar_Ch_06 : Array[1..200] of Int;   // Массив значений канала 6
      ar_Ch_07 : Array[1..200] of Int;   // Массив значений канала 7
      ar_Ch_08 : Array[1..200] of Int;   // Массив значений канала 8
      ar_Ch_09 : Array[1..200] of Int;   // Массив значений канала 9
      ar_Ch_10 : Array[1..200] of Int;   // Массив значений канала 10
      ar_Ramp : Array[1..200] of Int;   // Массив значений с пилой
      Ch_1 : Int;   // Текущее значение канала 1
      Ch_2 : Int;   // Текущее значение канала 2
      Ch_3 : Int;   // Текущее значение канала 3
      Ch_4 : Int;   // Текущее значение канала 4
      Ch_5 : Int;   // Текущее значение канала 5
      Ch_6 : Int;   // Текущее значение канала 6
      Ch_7 : Int;   // Текущее значение канала 7
      Ch_8 : Int;   // Текущее значение канала 8
      Ch_9 : Int;   // Текущее значение канала 9
      Ch_10 : Int;   // Текущее значение канала 10
   END_VAR
BEGIN
   ar_Ch_01[17] := 276;
END_DATA_BLOCK

FUNCTION "OSC" : Void   // FC500, STL
{ S7_Optimized_Access := 'FALSE' }
VERSION : 0.1
   VAR_TEMP
      CH_10 : Int;
      CH_09 : Int;
      CH_08 : Int;
      CH_07 : Int;
      CH_06 : Int;
      CH_05 : Int;
      CH_04 : Int;
      CH_03 : Int;
      CH_02 : Int;
      CH_01 : Int;
      TMP_DI : DInt;
      For_SIN : Int;
   END_VAR
BEGIN

REGION Network 1

   //      CALL  "OSC_BS_GP"
   //         Ch_01 :=#CH_01
   //         Ch_02 :=#CH_02
   //         Ch_03 :=#CH_03
   //         Ch_04 :=#CH_04
   //         Ch_05 :=#CH_05
   //         Ch_06 :=#CH_06
   //         Ch_07 :=#CH_07
   //         Ch_08 :=#CH_08
   //         Ch_09 :=#CH_09
   //         Ch_10 :=#CH_10

   //      CALL  "Bl_Spr_OE"
   //       Ch_01:=#CH_01
   //       Ch_02:=#CH_02
   //       Ch_03:=#CH_03
   //       Ch_04:=#CH_04
   //       Ch_05:=#CH_05
   //       Ch_06:=#CH_06
   //       Ch_07:=#CH_07
   //       Ch_08:=#CH_08
   //       Ch_09:=#CH_09
   //       Ch_10:=#CH_10

   //      CALL  FC   514
   //       Ch_01:=#CH_01
   //       Ch_02:=#CH_02
   //       Ch_03:=#CH_03
   //       Ch_04:=#CH_04
   //       Ch_05:=#CH_05
   //       Ch_06:=#CH_06
   //       Ch_07:=#CH_07
   //       Ch_08:=#CH_08
   //       Ch_09:=#CH_09
   //       Ch_10:=#CH_10


         L     "Temp".Radians;
         L     0.2;
         +R;
         T     "Temp".Radians;
         L     5000.0;
         >R;
         JNB   _002;

         L     0.0;
         T     "Temp".Radians;

   _002: NOP   0;

   //     ITD
   //      DTR
         L     "Temp".Radians;
         COS;
         L     1000.0;
         *R;
         TRUNC;
         T     #For_SIN;

         L     100.0;
         *R;


   //== Запись в массив оссциллографирования
         CALL  "Wr_OSC"
         ( Var_1  := #For_SIN,
           Var_2  := #CH_02,
           Var_3  := #CH_03,
           Var_4  := #CH_04,
           Var_5  := #CH_05,
           Var_6  := #CH_06,
           Var_7  := #CH_07,
           Var_8  := #CH_08,
           Var_9  := #CH_09,
           Var_10 := #CH_10
         );
END_REGION

REGION Network 2



         A(;
         L     "DB_OSC".Ramp;
         L     1;
         +I;
         T     "DB_OSC".Ramp;
         AN    OV;
         SAVE;
         CLR;
         A     BR;
         );
         A(;
         L     "DB_OSC".Ramp;
         L     5000;
         >I;
         );
         JNB   _001;
         L     0;
         T     "DB_OSC".Ramp;
   _001: NOP   0;
END_REGION
END_FUNCTION

FUNCTION "Wr_OSC" : Void   // FC505, STL
{ S7_Optimized_Access := 'FALSE' }
VERSION : 0.1
// Запись параметров в массив осцилографирования
// Версия 20-10-2014
   VAR_INPUT
      Var_1 : Int;
      Var_2 : Int;
      Var_3 : Int;
      Var_4 : Int;
      Var_5 : Int;
      Var_6 : Int;
      Var_7 : Int;
      Var_8 : Int;
      Var_9 : Int;
      Var_10 : Int;
   END_VAR
   VAR_TEMP
      Tmp_1 : DInt;
      Tmp_2 : DInt;
      Tmp_3 : DInt;
      Tmp_4 : DInt;
      Tmp_5 : DInt;
      Tmp_6 : DInt;
      Tmp_7 : DInt;
      Tmp_Ramp : DInt;
      Ramp : Int;
      Tmp_8 : DInt;
      Tmp_9 : DInt;
      Tmp_10 : DInt;
      RV : Int;
   END_VAR
BEGIN

REGION Network 1
   // 658619651
         A     %DB505.DBX1.0;
         FP    "OSC_Work";
         JNB   STRT;

         CALL  "Ini_Arr"
         ( Reg := 0
         );

   STRT: A     %DB505.DBX1.0;
         JNB   FIN;

   //---------------- Расчёт номера участка
         L     1;
         L     "DB_OSC".Cnt;
         +I;
         T     "DB_OSC".Cnt;
         L     50;
         >I;
         JNB   _NFR;

         L     1;
         T     "DB_OSC".Cnt;

         L     1;
         L     "DB_OSC".Ready;
         +I;
         T     "DB_OSC".Ready;
         L     4;
         >I;
         JNB   _NFR;

         L     1;
         T     "DB_OSC".Ready;

   _NFR: NOP   0;

   //------------------------------------
         L     "DB_OSC".cr_Addr_1;
         T     #Tmp_1;

         L     "DB_OSC".cr_Addr_2;
         T     #Tmp_2;

         L     "DB_OSC".cr_Addr_3;
         T     #Tmp_3;

         L     "DB_OSC".cr_Addr_4;
         T     #Tmp_4;

         L     "DB_OSC".cr_Addr_5;
         T     #Tmp_5;

         L     "DB_OSC".cr_Addr_6;
         T     #Tmp_6;

         L     "DB_OSC".cr_Addr_7;
         T     #Tmp_7;

         L     "DB_OSC".cr_Addr_8;
         T     #Tmp_8;

         L     "DB_OSC".cr_Addr_9;
         T     #Tmp_9;

         L     "DB_OSC".cr_Addr_10;
         T     #Tmp_10;

   //--------------------------------
   // Запись значений в блок данных
   //--------------------------------
         OPN   "DB_OSC";
         L     #Var_1;
         T     DBW [#Tmp_1];
         T     "DB_OSC".Ch_1;

         L     #Var_2;
         T     DBW [#Tmp_2];
         T     "DB_OSC".Ch_2;

         L     #Var_3;
         T     DBW [#Tmp_3];
         T     "DB_OSC".Ch_3;

         L     #Var_4;
         T     DBW [#Tmp_4];
         T     "DB_OSC".Ch_4;

         L     #Var_5;
         T     DBW [#Tmp_5];
         T     "DB_OSC".Ch_5;

         L     #Var_6;
         T     DBW [#Tmp_6];
         T     "DB_OSC".Ch_6;

         L     #Var_7;
         T     DBW [#Tmp_7];
         T     "DB_OSC".Ch_7;

         L     #Var_8;
         T     DBW [#Tmp_8];
         T     "DB_OSC".Ch_8;

         L     #Var_9;
         T     DBW [#Tmp_9];
         T     "DB_OSC".Ch_9;

         L     #Var_10;
         T     DBW [#Tmp_10];
         T     "DB_OSC".Ch_10;

   //------------------------------
   // Пересчёт адресов
   //------------------------------
         L     DINT#16;
         L     "DB_OSC".cr_Addr_1;
         +D;
         T     "DB_OSC".cr_Addr_1;

         L     DINT#16;
         L     "DB_OSC".cr_Addr_2;
         +D;
         T     "DB_OSC".cr_Addr_2;

         L     DINT#16;
         L     "DB_OSC".cr_Addr_3;
         +D;
         T     "DB_OSC".cr_Addr_3;

         L     DINT#16;
         L     "DB_OSC".cr_Addr_4;
         +D;
         T     "DB_OSC".cr_Addr_4;

         L     DINT#16;
         L     "DB_OSC".cr_Addr_5;
         +D;
         T     "DB_OSC".cr_Addr_5;

         L     DINT#16;
         L     "DB_OSC".cr_Addr_6;
         +D;
         T     "DB_OSC".cr_Addr_6;

         L     DINT#16;
         L     "DB_OSC".cr_Addr_7;
         +D;
         T     "DB_OSC".cr_Addr_7;

         L     DINT#16;
         L     "DB_OSC".cr_Addr_8;
         +D;
         T     "DB_OSC".cr_Addr_8;

         L     DINT#16;
         L     "DB_OSC".cr_Addr_9;
         +D;
         T     "DB_OSC".cr_Addr_9;

         L     DINT#16;
         L     "DB_OSC".cr_Addr_10;
         +D;
         T     "DB_OSC".cr_Addr_10;

         L     DINT#16;
         L     "DB_OSC".cr_Addr_Rmp;
         +D;
         T     "DB_OSC".cr_Addr_Rmp;

         L     "DB_OSC".Max_Addr;
         >D;
         JNB   _NAR;

         CALL  "Ini_Arr"
         ( Reg := 1
         );

   _NAR: NOP   0;

   FIN:  NOP   0;
END_REGION
END_FUNCTION

FUNCTION "Ini_Arr" : Void   // FC506, STL
{ S7_Optimized_Access := 'FALSE' }
VERSION : 0.0
// Инициализация параметров осцилографирования
// Версия: 16-10-2014
// Входные параметры:
//   Reg - режим работы программы
//     0 - Задать адреса набора 1 и очистить все массивы
//     1 - Задать адреса набора 1
//     2 - Задать адреса набора 2
   VAR_INPUT
      Reg : Int;
   END_VAR
   VAR_TEMP
      Addr : DInt;
   END_VAR
BEGIN

REGION Network 1: SCL network

   //--------------------------------------
   // Начальные адреса массивов
   //--------------------------------------
         L     DINT#448;
         T     "DB_OSC".cr_Addr_1;
         L     DINT#3648;
         T     "DB_OSC".cr_Addr_2;
         L     DINT#6848;
         T     "DB_OSC".cr_Addr_3;
         L     DINT#10048;
         T     "DB_OSC".cr_Addr_4;
         L     DINT#13248;
         T     "DB_OSC".cr_Addr_5;
         L     DINT#16448;
         T     "DB_OSC".cr_Addr_6;
         L     DINT#19648;
         T     "DB_OSC".cr_Addr_7;
         L     DINT#22848;
         T     "DB_OSC".cr_Addr_8;
         L     DINT#26048;
         T     "DB_OSC".cr_Addr_9;
         L     DINT#29248;
         T     "DB_OSC".cr_Addr_10;
         L     DINT#32448;
         T     "DB_OSC".cr_Addr_Rmp;

         L     DINT#35632;
         T     "DB_OSC".Max_Addr;

   //--------------------------------------
   // Первая инициализация
   //--------------------------------------
         L     #Reg;
         L     0;
         ==I;
         JCN   A7d1;

   //--------------------------------------
   // Очистка массивов
   //--------------------------------------
         L     0;
         T     "DB_OSC".Ready;
         T     "DB_OSC".Cnt;
         T     "DB_OSC".Ramp;

         L     "DB_OSC".cr_Addr_1;
         T     #Addr;

   A7d3: L     #Addr;
         L     "DB_OSC".Max_Addr;
         <=D;
         JCN   A7d1;

         OPN   "DB_OSC";
         L     DINT#0;
         T     DBW [#Addr];

         L     #Addr;
         L     DINT#16;
         +D;
         T     #Addr;
         JU    A7d3;

   A7d1: NOP   0;

         SAVE;
         CLR;
END_REGION
END_FUNCTION

FUNCTION "OSC_BS_GP" : Void   // FC511, STL
{ S7_Optimized_Access := 'FALSE' }
VERSION : 0.1
   VAR_OUTPUT
      Ch_01 : Int;   // Данные для канала 1
      Ch_02 : Int;   // Данные для канала 2
      Ch_03 : Int;   // Данные для канала 3
      Ch_04 : Int;   // Данные для канала 4
      Ch_05 : Int;   // Данные для канала 5
      Ch_06 : Int;   // Данные для канала 6
      Ch_07 : Int;   // Данные для канала 7
      Ch_08 : Int;   // Данные для канала 8
      Ch_09 : Int;   // Данные для канала 9
      Ch_10 : Int;   // Данные для канала 10
   END_VAR
   VAR_TEMP
      Tmp_DI : DInt;
   END_VAR
BEGIN

REGION Network 1

   //======================== #CH_01
         L     "SU".su_Iq_M1H_fs;
         L     10.0;
         *R;
         RND;
         T     #Tmp_DI;
         L     <??.?>;
         T     #Ch_01;

   //======================== #CH_02
         L     "SU".su_W_M1H_fs;
         L     10.0;
         *R;
         RND;
         T     #Tmp_DI;
         L     <??.?>;
         T     #Ch_02;

   //======================== #CH_03
         L     "SU".su_LH;
         L     10.0;
         *R;
         RND;
         T     #Tmp_DI;
         L     <??.?>;
         T     #Ch_03;

   //======================== #CH_04
         L     "SU".su_LC;
         L     10.0;
         *R;
         RND;
         T     #Tmp_DI;
         L     <??.?>;
         T     #Ch_04;

   //======================== #CH_05
         L     "SU".su_W_S_fs;
         L     10.0;
         *R;
         RND;
         T     #Tmp_DI;
         L     <??.?>;
         T     #Ch_05;

   //======================== #CH_06
         L     "SU".su_Job_C;
         L     DINT#10;
         /D;
         T     #Tmp_DI;
         L     <??.?>;
         T     #Ch_06;


   //      L     "SU".su_Iq_S_fs
   //      L     "SU".su_W_C_fs
   ///      L     1.000000e+001
   //      *R
   //      RND
   //      T     #Tmp_DI
   //      L     LW     2

   //======================== #CH_07
         L     "Work".ug_Pov_Tk;
         T     #Ch_07;

   //      L     "SU".su_LH
   //      L     1.000000e+001
   //      *R
   //      RND
   //      T     #Tmp_DI
   //      L     LW     2

   //======================== #CH_08
         L     "Work".Reg_WC;
         L     100;
         *I;
         T     #Ch_08;

         A     "AP".ap_Gudok;
         JNB   _NGD;

         L     -100;
         T     #Ch_08;

   _NGD: NOP   0;

         A     "AP".ap_ODK;
         JNB   _NOD;

         L     700;
         T     #Ch_08;

   _NOD: NOP   0;

   //      L     "SU".su_LC
   //      L     1.000000e+001
   //      *R
   //      RND
   //     T     #Tmp_DI
   //      L     LW     2

   //======================== #CH_09
         L     "BD".Mas_Basket;
         L     10.0;
         *R;
         RND;
         T     #Tmp_DI;
         L     <??.?>;
         T     #Ch_09;

   //======================== #CH_10
   //      L     "SU".su_Iq_S_fs
         L     "Work".ABS_H;
         L     10.0;
         *R;
         RND;
         T     #Tmp_DI;
         L     <??.?>;
         T     #Ch_10;
END_REGION
END_FUNCTION

FUNCTION "FC514" : Void   // FC514, STL
TITLE = Блок сопряжения осц-фа для ОЭ
{ S7_Optimized_Access := 'FALSE' }
VERSION : 0.1
   VAR_OUTPUT
      Ch_01 : Int;   // Данные для канала 1
      Ch_02 : Int;   // Данные для канала 2
      Ch_03 : Int;   // Данные для канала 3
      Ch_04 : Int;   // Данные для канала 4
      Ch_05 : Int;   // Данные для канала 5
      Ch_06 : Int;   // Данные для канала 6
      Ch_07 : Int;   // Данные для канала 7
      Ch_08 : Int;   // Данные для канала 8
      Ch_09 : Int;   // Данные для канала 9
      Ch_10 : Int;   // Данные для канала 10
   END_VAR
   VAR_TEMP
      Tmp_DI : DInt;
   END_VAR
BEGIN

REGION Network 1

   //======================== #CH_01
         L     "SU".su_Iq_M1H_fs;
         L     10.0;
         *R;
         RND;
         T     #Tmp_DI;
         L     <??.?>;
         T     #Ch_01;

   //======================== #CH_02
         L     "SU".su_W_M1H_fs;
         L     10.0;
         *R;
         RND;
         T     #Tmp_DI;
         L     <??.?>;
         T     #Ch_02;

   //======================== #CH_03
         L     "SU".su_Iq_S_fs;
         L     10.0;
         *R;
         RND;
         T     #Tmp_DI;
         L     <??.?>;
         T     #Ch_03;

   //======================== #CH_04
         L     "SU".su_W_S_fs;
         L     10.0;
         *R;
         RND;
         T     #Tmp_DI;
         L     <??.?>;
         T     #Ch_04;

   //======================== #CH_05
         L     "SU".su_Iq_C_fs;
         L     10.0;
         *R;
         RND;
         T     #Tmp_DI;
         L     <??.?>;
         T     #Ch_05;

   //======================== #CH_06
         L     "SU".su_W_C_fs;
         L     10.0;
         *R;
         RND;
         T     #Tmp_DI;
         L     <??.?>;
         T     #Ch_06;

   //======================== #CH_07
         L     "SU".su_LH;
         L     10.0;
         *R;
         RND;
         T     #Tmp_DI;
         L     <??.?>;
         T     #Ch_07;

   //======================== #CH_08
         L     "SU".su_LC;
         L     10.0;
         *R;
         RND;
         T     #Tmp_DI;
         L     <??.?>;
         T     #Ch_08;

   //======================== #CH_09
         L     "SU".su_Iq_C_fs;
         L     10.0;
         *R;
         RND;
         T     #Tmp_DI;
         L     <??.?>;
         T     #Ch_09;

   //======================== #CH_10
         L     "BD".Mas_TS_cr;
         L     10.0;
         *R;
         RND;
         T     #Tmp_DI;
         L     <??.?>;
         T     #Ch_10;
END_REGION
END_FUNCTION

ORGANIZATION_BLOCK "Main"   // OB1, LAD
TITLE = "Main Program Sweep (Cycle)"
{ S7_Optimized_Access := 'FALSE' }
VERSION : 0.1
   VAR_TEMP
      OB1_EV_CLASS : Byte;   // Bits 0-3 = 1 (Coming event), Bits 4-7 = 1 (Event class 1)
      OB1_SCAN_1 : Byte;   // 1 (Cold restart scan 1 of OB 1), 3 (Scan 2-n of OB 1)
      OB1_PRIORITY : Byte;   // Priority of OB Execution
      OB1_OB_NUMBR : Byte;   // 1 (Organization block 1, OB1)
      OB1_RESERVED_1 : Byte;   // Reserved for system
      OB1_RESERVED_2 : Byte;   // Reserved for system
      OB1_PREV_CYCLE : Int;   // Cycle time of previous OB1 scan (milliseconds)
      OB1_MIN_CYCLE : Int;   // Minimum cycle time of OB1 (milliseconds)
      OB1_MAX_CYCLE : Int;   // Maximum cycle time of OB1 (milliseconds)
      OB1_DATE_TIME : Date_And_Time;   // Date and time OB1 started
   END_VAR
BEGIN
END_ORGANIZATION_BLOCK

ORGANIZATION_BLOCK "CYC_INT5"   // OB35, STL
TITLE = "Cyclic Interrupt"
{ S7_Optimized_Access := 'FALSE' }
VERSION : 0.1
   VAR_TEMP
      OB35_EV_CLASS : Byte;   // Bits 0-3 = 1 (Coming event), Bits 4-7 = 1 (Event class 1)
      OB35_STRT_INF : Byte;   // 16#36 (OB 35 has started)
      OB35_PRIORITY : Byte;   // Priority of OB Execution
      OB35_OB_NUMBR : Byte;   // 35 (Organization block 35, OB35)
      OB35_RESERVED_1 : Byte;   // Reserved for system
      OB35_RESERVED_2 : Byte;   // Reserved for system
      OB35_PHASE_OFFSET : Word;   // Phase offset (msec)
      OB35_RESERVED_3 : Int;   // Reserved for system
      OB35_EXC_FREQ : Int;   // Frequency of execution (msec)
      OB35_DATE_TIME : Date_And_Time;   // Date and time OB35 started
   END_VAR
BEGIN

REGION Network 1
         CALL  "OSC";
END_REGION
END_ORGANIZATION_BLOCK

// ===== PLC "PLC_2"  CPU 1512SP-1 PN =====

VAR_GLOBAL   // PLC tag table "Merkers"
   "OSC_Work" AT %M20.5 : Bool;
END_VAR

DATA_BLOCK "Temp"   // DB1
{ S7_Optimized_Access := 'FALSE' }
VERSION : 0.1
   VAR
      Radians : Real;
      Ramp : Real;
      Square : Real;
      TriangleUp : Real;
      If_Up : Bool;   // признак прироста треугольника вверх
   END_VAR
BEGIN
END_DATA_BLOCK

DATA_BLOCK "SU"   // DB101
{ S7_Optimized_Access := 'FALSE' }
VERSION : 0.1
   VAR
      su_Uac_6kV : Real;   // Действующее линейное напряжение AC на входе ЯВВ, В
      Spare_4_0 : Int;   // Резерв
      su_Fan_MD_QF1 : Bool;   // Автомат вентиляторов QF1 (0-выкл,1-вкл)
      su_Fan_MD_QF2 : Bool;   // Автомат вентиляторов QF2 (0-выкл,1-вкл)
      su_Fan_MD_QF3 : Bool;   // Автомат вентиляторов QF3 (0-выкл,1-вкл)
      su_Fan_MD_QF4 : Bool;   // Автомат вентиляторов QF4 (0-выкл,1-вкл)
      su_Fan_M1_ON : Bool;   // Контактор вентилятора КМ1 (0-выкл,1-вкл)
      su_Fan_M2_ON : Bool;   // Контактор вентилятора КМ2 (0-выкл,1-вкл)
      su_Fan_M6_ON : Bool;   // Контактор вентилятора КМ6 (0-выкл,1-вкл)
      su_Fan_M7_ON : Bool;   // Контактор вентилятора КМ7 (0-выкл,1-вкл)
      su_Fan_M8_ON : Bool;   // Контактор вентилятора КМ8 (0-выкл,1-вкл)
      su_Temp_ok : Bool;   // Температура в норме (0-выкл,1-вкл)
      su_Fan_MD_Ready : Bool;   // Готовность вентиляции ГП (0-выкл,1-вкл)
      su_Fan_M3_ON : Bool;   // Контактор вентилятора КМ3 (0-выкл,1-вкл)
      su_Fan_M4_ON : Bool;   // Контактор вентилятора КМ4 (0-выкл,1-вкл)
      su_Fan_M5_ON : Bool;   // Контактор вентилятора КМ5 (0-выкл,1-вкл)
      su_LH : Real;   // Длина подъемного каната, м
      su_LC : Real;   // Длина выдвижения рукояти, м
      su_OHRVD_AF : Bool;   // Ограничение хода рукояти. При выдвижении (0-ограничение выкл,1-ограничение)
      su_OHRVT_AF : Bool;   // Ограничение хода рукояти. При втягивании (0-ограничение выкл,1-ограничение)
      su_LC_Reset : Bool;   // Обнулить знчение энкодера напора (1-обнулить)
      su_OPK_AF : Bool;   // Ограничение подъема ковша (0-ограничение выкл, 1-ограничение)
      su_LH_Reset : Bool;   // Обнулить знчение энкодера подъема (1-обнулить)
      su_Field_Reduction : Bool;   // Ослабление поля (0-выкл,1-вкл)
      su_Field_Forcing : Bool;   // Форсировка поля (0-выкл,1-вкл)
      su_Autobrake_ON : Bool;   // Подхват тормозов (0-выкл,1-вкл)
      su_Brake_H : Bool;   // Тормоза привода подъема (1–расторможен,0–заторможен)
      su_Brake_C : Bool;   // Тормоза привода напора (1–расторможен,0–заторможен)
      su_Brake_S : Bool;   // Тормоза привода поворота (1–расторможен,0–заторможен)
      su_Brake_P : Bool;   // Тормоза привода хода левого (1–расторможен,0–заторможен)
      su_Brake_P_R : Bool;   // Тормоза привода хода правого (1–расторможен,0–заторможен)
      su_All_Protect : Bool;   // Автоматические защиты (0-выкл,1–вкл)
      su_BOS_Connect : Bool;   // Связь с БОС (0-связь есть,1-связи нет)
      su_Job_Limit : Bool;   // Уровень ограничения задания (0-задание 100%,1-задание 70%)
      su_Blocking_1 : Bool;   // Блокировка 1 Защита выше напорного вала (1-вкл,0-выкл)
      su_Blocking_2 : Bool;   // Блокировка 2 Защита при збросе ковша (1-вкл,0-выкл)
      su_Blocking_3 : Bool;   // Блокировка 3 Ограничение хода рукояти (1-вкл,0-выкл)
      su_Blocking_4 : Bool;   // Блокировка 4 Ограничение подъема ковша (1-вкл,0-выкл)
      su_Blocking_5 : Bool;   // Блокировка 5 Ограничение боковых нагрузок при черпании(1-вкл,0-выкл)
      su_Blocking_6 : Bool;   // Блокировка 6 Ограничение боковых нагрузок при работе с негабаритами(1-вкл,0-вык
      su_Blocking_7 : Bool;   // Блокировка 7 Передняя кромка(1-вкл,0-выкл)
      su_Blocking_8 : Bool;   // Блокировка 8 Защита от заброса стрелы(1-вкл,0-выкл)
      su_Blocking_9 : Bool;   // Блокировка 9 Ограничение длины разматывания подъемного каната (1-вкл,0-выкл)
      su_Enc_C_Connect : Bool;   // Энкодер напора подключен (1-связь есть,0-связи нет)
      su_Enc_H_Connect : Bool;   // Энкодер подъема подключен (1-связь есть,0-связи нет)
      Spare_19_3 : Bool;   // Резерв
      Spare_19_4 : Bool;   // Резерв
      Spare_19_5 : Bool;   // Резерв
      Spare_19_6 : Bool;   // Резерв
      Spare_19_7 : Bool;   // Резерв
      su_Job_H : DInt := DINT#0;   // Задание для привода подъема
      su_Job_S : DInt := DINT#0;   // Задание для привода поворота
      Spare_28_0 : Int;   // Резерв
      su_Excav : Bool;   // Режим "Экскавация" (1-вкл,0-выкл)
      su_Prop : Bool;   // Режим "Ход" (1-вкл,0-выкл)
      su_Work_S : Bool;   // Привод поворота расторможен (1-вкл,0-выкл)
      su_Work_C : Bool;   // Привод напора расторможен (1-вкл,0-выкл)
      su_Work_H : Bool;   // Привод подъема расторможен (1-вкл,0-выкл)
      su_Ready_S : Bool;   // Разрешение растормозить привод поворота (1-вкл,0-выкл)
      su_Fan_Prop : Bool;   // Вентиляторы двигателей хода (1-вкл,0-выкл)
      su_AR_Mode_Work : Bool;   // Активные выпрямители в режиме "Работа" (1-вкл,0-выкл)
      su_Ctrl_Is : Bool;   // Контроль изоляции (1-вкл,0-выкл)
      su_Ctrl_Ladder : Bool;   // Контроль положения лестницы (1-вкл,0-выкл)
      su_Relay_Alarm_ON : Bool;   // Реле включения аварии (1-вкл,0-выкл)
      su_Relay_CtrlC : Bool;   // Реле включения цепей управления (1-вкл,0-выкл)
      su_Ctrl_Breaker : Bool;   // Контроль состояния вводных автоматов (1-вкл,0-выкл)
      su_Limit_Switch : Bool;   // Конечные выключатели шкафов управления (1-вкл,0-выкл)
      su_Ready_P : Bool;   // Разрешение растормозить привод хода (1-вкл,0-выкл)
      su_Fan_Mot : Bool;   // Вентиляция машин (1-вкл,0-выкл)
      su_Work_P : Bool;   // Привод хода расторможен (1-вкл,0-выкл)
      su_Lubr : Bool;   // Смазка редукторов поворота (1-вкл,0-выкл)
      su_BUP_StartUp_ARm : Bool;   // Блок управления в режиме инициализации (1-вкл,0-выкл)
      su_BUP_ON_ARm : Bool;   // Блок управления в работе, управляющие импульсы поданы (1-вкл,0-выкл)
      su_BUP_StartUp_ARs1 : Bool;   // Блок управления в режиме инициализации (1-вкл,0-выкл)
      su_BUP_ON_ARs1 : Bool;   // Блок управления в работе, управляющие импульсы поданы (1-вкл,0-выкл)
      su_BUP_StartUp_ARs2 : Bool;   // Блок управления в режиме инициализации (1-вкл,0-выкл)
      su_BUP_ON_ARs2 : Bool;   // Блок управления в работе, управляющие импульсы поданы (1-вкл,0-выкл)
      su_BUP_StartUp_ARs3 : Bool;   // Блок управления в режиме инициализации (1-вкл,0-выкл)
      su_BUP_ON_ARs3 : Bool;   // Блок управления в работе, управляющие импульсы поданы (1-вкл,0-выкл)
      su_Magnet_M1H : Bool;   // Двигатель намагничен (1-вкл,0-выкл)
      su_BUP_StartUp_Hm : Bool;   // Блок управления в режиме инициализации (1-вкл,0-выкл)
      su_BUP_ON_Hm : Bool;   // Блок управления в работе, управляющие импульсы поданы (1-вкл,0-выкл)
      su_Magnet_M2H : Bool;   // Двигатель намагничен (1-вкл,0-выкл)
      su_BUP_StartUp_Hs : Bool;   // Блок управления в режиме инициализации (1-вкл,0-выкл)
      su_BUP_ON_Hs : Bool;   // Блок управления в работе, управляющие импульсы поданы (1-вкл,0-выкл)
      su_Magnet_MC : Bool;   // Двигатель намагничен (1-вкл,0-выкл)
      su_BUP_StartUp_C : Bool;   // Блок управления в режиме инициализации (1-вкл,0-выкл)
      su_BUP_ON_C : Bool;   // Блок управления в работе, управляющие импульсы поданы (1-вкл,0-выкл)
      su_Magnet_M1S : Bool;   // Двигатель намагничен (1-вкл,0-выкл)
      su_BUP_StartUp_Sm : Bool;   // Блок управления в режиме инициализации (1-вкл,0-выкл)
      su_BUP_ON_Sm : Bool;   // Блок управления в работе, управляющие импульсы поданы (1-вкл,0-выкл)
      su_Magnet_M2S : Bool;   // Двигатель намагничен (1-вкл,0-выкл)
      su_BUP_StartUp_Ss1 : Bool;   // Блок управления в режиме инициализации (1-вкл,0-выкл)
      su_BUP_ON_Ss1 : Bool;   // Блок управления в работе, управляющие импульсы поданы (1-вкл,0-выкл)
      su_Magnet_M3S : Bool;   // Двигатель намагничен (1-вкл,0-выкл)
      su_BUP_StartUp_Ss2 : Bool;   // Блок управления в режиме инициализации (1-вкл,0-выкл)
      su_BUP_ON_Ss2 : Bool;   // Блок управления в работе, управляющие импульсы поданы (1-вкл,0-выкл)
      su_Magnet_M4S : Bool;   // Двигатель намагничен (1-вкл,0-выкл)
      su_BUP_StartUp_Ss3 : Bool;   // Блок управления в режиме инициализации (1-вкл,0-выкл)
      su_BUP_ON_Ss3 : Bool;   // Блок управления в работе, управляющие импульсы поданы (1-вкл,0-выкл)
      su_Magnet_M1P : Bool;   // Двигатель намагничен (1-вкл,0-выкл)
      su_BUP_StartUp_C_P : Bool;   // Блок управления в режиме инициализации (1-вкл,0-выкл)
      su_BUP_ON_C_P : Bool;   // Блок управления в работе, управляющие импульсы поданы (1-вкл,0-выкл)
      su_Magnet_M2P : Bool;   // Двигатель намагничен (1-вкл,0-выкл)
      su_BUP_StartUp_S_P : Bool;   // Блок управления в режиме инициализации (1-вкл,0-выкл)
      su_BUP_ON_S_P : Bool;   // Блок управления в работе, управляющие импульсы поданы (1-вкл,0-выкл)
      Spare_36_5 : Bool;   // Резерв
      Spare_36_6 : Bool;   // Резерв
      Spare_36_7 : Bool;   // Резерв
      Spare_37_B : Byte;   // Резерв
      su_I_ARm : Real;   // Действующий ток, А
      su_Ud_ARm : Real;   // Напряжение звена постоянного тока, В
      su_Ia_ARm : Real;   // Амплитудный активный ток выпрямителя, А
      su_Ir_ARm : Real;   // Амплитудный индуктивный ток выпрямителя, А
      su_fs_ARm : Real;   // Частота сети
      su_Us_ARm : Real;   // Амплитудное напряжение на входе выпрямителя
      su_Pa_ARm : Real;   // Активная мощность выпрямителя
      su_I_ARs1 : Real;   // Действующий ток, А
      su_Ud_ARs1 : Real;   // Напряжение звена постоянного тока, В
      su_Ia_ARs1 : Real;   // Амплитудный активный ток выпрямителя, А
      su_Ir_ARs1 : Real;   // Амплитудный индуктивный ток выпрямителя, А
      su_fs_ARs1 : Real;   // Частота сети
      su_Us_ARs1 : Real;   // Амплитудное напряжение на входе выпрямителя
      su_Pa_ARs1 : Real;   // Активная мощность выпрямителя
      su_Job_I_ARs1 : Real;   // Задание на регулятор тока ведомого выпрямителя
      su_I_ARs2 : Real;   // Действующий ток, А
      su_Ud_ARs2 : Real;   // Напряжение звена постоянного тока, В
      su_Ia_ARs2 : Real;   // Амплитудный активный ток выпрямителя, А
      su_Ir_ARs2 : Real;   // Амплитудный индуктивный ток выпрямителя, А
      su_fs_ARs2 : Real;   // Частота сети
      su_Us_ARs2 : Real;   // Амплитудное напряжение на входе выпрямителя
      su_Pa_ARs2 : Real;   // Активная мощность выпрямителя
      su_Job_I_ARs2 : Real;   // Задание на регулятор тока ведомого выпрямителя
      su_I_ARs3 : Real;   // Действующий ток, А
      su_Ud_ARs3 : Real;   // Напряжение звена постоянного тока, В
      su_Ia_ARs3 : Real;   // Амплитудный активный ток выпрямителя, А
      su_Ir_ARs3 : Real;   // Амплитудный индуктивный ток выпрямителя, А
      su_fs_ARs3 : Real;   // Частота сети
      su_Us_ARs3 : Real;   // Амплитудное напряжение на входе выпрямителя
      su_Pa_ARs3 : Real;   // Активная мощность выпрямителя
      su_Job_I_ARs3 : Real;   // Задание на регулятор тока ведомого выпрямителя
      su_I_M1H : Real;   // Действующий ток статора, А
      su_Ud_Hm : Real;   // Напряжение звена постоянного тока, В
      su_Id_M1H : Real;   // Ток намагничивания статора, А
      su_Iq_M1H : Real;   // Активный ток статора, А
      su_W_M1H : Real;   // Скорость, рад/с
      su_Psi2_M1H : Real;   // Поток ротора, Вб
      su_U_M1H : Real;   // Фазное напряжение двигателя, В
      su_JobW_Hm : Real;   // Задание на скорость, ед
      su_I_M2H : Real;   // Действующий ток статора, А
      su_Ud_Hs : Real;   // Напряжение звена постоянного тока, В
      su_Id_M2H : Real;   // Ток намагничивания статора, А
      su_Iq_M2H : Real;   // Активный ток статора, А
      su_W_M2H : Real;   // Скорость, рад/с
      su_Psi2_M2H : Real;   // Поток ротора, Вб
      su_U_M2H : Real;   // Фазное напряжение двигателя, В
      su_JobW_Hs : Real;   // Задание на скорость, ед
      su_I_MC : Real;   // Действующий ток статора, А
      su_Ud_C : Real;   // Напряжение звена постоянного тока, В
      su_Id_MC : Real;   // Ток намагничивания статора, А
      su_Iq_MC : Real;   // Активный ток статора, А
      su_W_MC : Real;   // Скорость, рад/с
      su_Psi2_MC : Real;   // Поток ротора, Вб
      su_U_MC : Real;   // Фазное напряжение двигателя, В
      su_JobW_C : Real;   // Задание на скорость, ед
      su_I_M1S : Real;   // Действующий ток статора, А
      su_Ud_Sm : Real;   // Напряжение звена постоянного тока, В
      su_Id_M1S : Real;   // Ток намагничивания статора, А
      su_Iq_M1S : Real;   // Активный ток статора, А
      su_W_M1S : Real;   // Скорость, рад/с
      su_Psi2_M1S : Real;   // Поток ротора, Вб
      su_U_M1S : Real;   // Фазное напряжение двигателя, В
      su_JobW_Sm : Real;   // Задание на скорость, ед
      su_I_M2S : Real;   // Действующий ток статора, А
      su_Ud_Ss1 : Real;   // Напряжение звена постоянного тока, В
      su_Id_M2S : Real;   // Ток намагничивания статора, А
      su_Iq_M2S : Real;   // Активный ток статора, А
      su_W_M2S : Real;   // Скорость, рад/с
      su_Psi2_M2S : Real;   // Поток ротора, Вб
      su_U_M2S : Real;   // Фазное напряжение двигателя, В
      su_JobW_Ss1 : Real;   // Задание на скорость, ед
      Spare_322_0 : Real;   // Резерв
      su_State_H1 : Bool;   // Готовность преобразователя подъема 1 (0-авария,1-готов)
      su_State_H2 : Bool;   // Готовность преобразователя подъема 2 (0-авария,1-готов)
      su_State_C : Bool;   // Готовность преобразователя напора (0-авария,1-готов)
      su_State_P1 : Bool;   // Готовность преобразователя хода 1 (0-авария,1-готов)
      su_State_P2 : Bool;   // Готовность преобразователя хода 2 (0-авария,1-готов)
      su_State_S1 : Bool;   // Готовность преобразователя поворота 1 (0-авария,1-готов)
      su_Overheat_TS : Bool;   // Перегрев силового трансформатора (0-авария,1-готов)
      su_GB_Charge : Bool;   // Блок заряда аккумуляторов (0-авария,1-готов)
      su_Relay_K4 : Bool;   // Реле К4 резерв (0-выкл,1-вкл)
      su_Relay_K3 : Bool;   // Реле К3, готовность блоков сброса (0-выкл,1-вкл)
      su_Relay_K2 : Bool;   // Реле К2 включение ВВ контактора (0-выкл,1-вкл)
      su_State_AR1 : Bool;   // Готовность активного выпрямителя 1 (0-авария,1-готов)
      su_State_AR2 : Bool;   // Готовность активного выпрямителя 2 (0-авария,1-готов)
      su_State_AR3 : Bool;   // Готовность активного выпрямителя 3 (0-авария,1-готов)
      su_State_Chop1 : Bool;   // Блок сброс 1 (0-авария,1-готов)
      su_State_Chop2 : Bool;   // Блок сброс 2 (0-авария,1-готов)
      su_Relay_K7 : Bool;   // Реле К7 резерв (0-выкл,1-вкл)
      su_Relay_K6 : Bool;   // Реле К6 резерв (0-выкл,1-вкл)
      su_State_AR4 : Bool;   // Готовность активного выпрямителя 4 (0-авария,1-готов)
      su_Relay_K5 : Bool;   // Реле К5 резерв (0-выкл,1-вкл)
      su_Relay_K1 : Bool;   // Реле К1 включение готовности преобразователей ГП (0-выкл,1-вкл)
      su_Vent_MD : Bool;   // Вентиляция главных приводов (0-выкл,1-вкл)
      su_HV_Contactor_ON : Bool;   // ВВ контактор включен (0-выкл,1-вкл)
      su_State_S2 : Bool;   // Готовность преобразователя поворота 2 (0-авария,1-готов)
      su_State_S3 : Bool;   // Готовность преобразователя поворота 3 (0-авария,1-готов)
      su_State_S4 : Bool;   // Готовность преобразователя поворота 4 (0-авария,1-готов)
      Spare_329_2 : Bool;   // Резерв
      Spare_329_3 : Bool;   // Резерв
      Spare_329_4 : Bool;   // Резерв
      Spare_329_5 : Bool;   // Резерв
      Spare_329_6 : Bool;   // Резерв
      Spare_329_7 : Bool;   // Резерв
      su_BOS_Enc_H : Int;   // Значение БОСЭ механизма подъема (1 оборот 2^10 бит)
      su_BOS_Enc_C : Int;   // Значение БОСЭ механизма напора (1 оборот 2^10 бит)
      su_MD_OFF : Bool;   // Отключение главных приводов (0-выкл,1-вкл)
      su_VH : Real;   // Линейная скорость подъема
      su_VC : Real;   // Линейная скорость напора
      su_Job_C : DInt := DINT#0;   // Задание для привода напора
      su_Ia_PowerT : Real;   // Ток в фазе А первичной обмотки силового трансформатора, А
      su_Ib_PowerT : Real;   // Ток в фазе В первичной обмотки силового трансформатора, А
      su_I_M3S : Real;   // Действующий ток статора, А
      su_Ud_Ss2 : Real;   // Напряжение звена постоянного тока, В
      su_Id_M3S : Real;   // Ток намагничивания статора, А
      su_Iq_M3S : Real;   // Активный ток статора, А
      su_W_M3S : Real;   // Скорость, рад/с
      su_Psi2_M3S : Real;   // Поток ротора, Вб
      su_U_M3S : Real;   // Фазное напряжение двигателя, В
      su_JobW_Ss2 : Real;   // Задание на скорость, ед
      su_I_M4S : Real;   // Действующий ток статора, А
      su_Ud_Ss3 : Real;   // Напряжение звена постоянного тока, В
      su_Id_M4S : Real;   // Ток намагничивания статора, А
      su_Iq_M4S : Real;   // Активный ток статора, А
      su_W_M4S : Real;   // Скорость, рад/с
      su_Psi2_M4S : Real;   // Поток ротора, Вб
      su_U_M4S : Real;   // Фазное напряжение двигателя, В
      su_JobW_Ss3 : Real;   // Задание на скорость, ед
      su_I_M1P : Real;   // Действующий ток статора, А
      su_Ud_C_P : Real;   // Напряжение звена постоянного тока, В
      su_Id_M1P : Real;   // Ток намагничивания статора, А
      su_Iq_M1P : Real;   // Активный ток статора, А
      su_W_M1P : Real;   // Скорость, рад/с
      su_Psi2_M1P : Real;   // Поток ротора, Вб
      su_U_M1P : Real;   // Фазное напряжение двигателя, В
      su_JobW_C_P : Real;   // Задание на скорость, ед
      su_I_M2P : Real;   // Действующий ток статора, А
      su_Ud_S_P : Real;   // Напряжение звена постоянного тока, В
      su_Id_M2P : Real;   // Ток намагничивания статора, А
      su_Iq_M2P : Real;   // Активный ток статора, А
      su_W_M2P : Real;   // Скорость, рад/с
      su_Psi2_M2P : Real;   // Поток ротора, Вб
      su_U_M2P : Real;   // Фазное напряжение двигателя, В
      su_JobW_S_P : Real;   // Задание на скорость, ед
      su_BUARm_ID : Int;   // Номер блока активного выпрямителя ведущего
      su_BUARs1_ID : Int;   // Номер блока активного выпрямителя ведомого 1
      su_BUARs2_ID : Int;   // Номер блока активного выпрямителя ведомого 2
      su_BUARs3_ID : Int;   // Номер блока активного выпрямителя ведомого 3
      su_Type_AR : Int;   // Текущий тип преобразователя
      su_BUP_Hm_ID : Int;   // Номер БУПа привода подъема ведущего
      su_BUP_Hs_ID : Int;   // Номер БУПа привода подъема ведомого
      su_BUP_C_ID : Int;   // Номер БУПа привода напора
      su_BUP_Sm_ID : Int;   // Номер БУПа привода поворота ведущего
      su_BUP_Ss1_ID : Int;   // Номер БУПа привода поворота ведомого 1
      su_BUP_Ss2_ID : Int;   // Номер БУПа привода поворота ведомого 2
      su_BUP_Ss3_ID : Int;   // Номер БУПа привода поворота ведомого 3
      su_BUP_CP_ID : Int;   // Номер БУПа привода напора-хода
      su_BUP_SP_ID : Int;   // Номер БУПа привода поворота-хода
      su_Type_Pr : Int;   // Текущий тип привода
      su_Temp_ARm : Int;   // Средняя температура активного выпрямителя ведущего
      su_Temp_ARs1 : Int;   // Средняя температура активного выпрямителя ведомого 1
      su_Temp_ARs3 : Int;   // Средняя температура активного выпрямителя ведомого 2
      su_Temp_ARs2 : Int;   // Средняя температура активного выпрямителя ведомого 3
      su_Temp_Hm : Int;   // Средняя температура преобразователя подъема ведущего
      su_Wr_M1H : Int;   // Электрическая скорость ротора M1H (показания датчика, рад/с)
      su_Temp_Hs : Int;   // Средняя температура преобразователя подъема ведомого
      su_Wr_M2H : Int;   // Электрическая скорость ротора M2H (показания датчика, рад/с)
      su_Temp_C : Int;   // Средняя температура преобразователя напора
      su_Wr_MC : Int;   // Электрическая скорость ротора MC (показания датчика, рад/с)
      su_Temp_Sm : Int;   // Средняя температура преобразователя поворота ведущего
      su_Wr_M1S : Int;   // Электрическая скорость ротора M1S (показания датчика, рад/с)
      su_Temp_Ss1 : Int;   // Средняя температура преобразователя поворота ведомого 1
      su_Wr_M2S : Int;   // Электрическая скорость ротора M2S (показания датчика, рад/с)
      su_Temp_Ss2 : Int;   // Средняя температура преобразователя поворота ведомого 2
      su_Wr_M3S : Int;   // Электрическая скорость ротора M3S (показания датчика, рад/с)
      su_Temp_Ss3 : Int;   // Средняя температура преобразователя поворота ведомого 3
      su_Wr_M4S : Int;   // Электрическая скорость ротора M4S (показания датчика, рад/с)
      su_Temp_C_P : Int;   // Средняя температура преобразователя напора-хода
      su_Wr_M1P : Int;   // Электрическая скорость ротора M1P (показания датчика, рад/с)
      su_Temp_S_P : Int;   // Средняя температура преобразователя поворота-хода
      su_Wr_M2P : Int;   // Электрическая скорость ротора M2P (показания датчика, рад/с)
      su_I_M1H_fs : Real;   // Действующий ток статора, A (быстрое значение)
      su_Id_M1H_fs : Real;   // Ток намагничивания статора, А (быстрое значение)
      su_Iq_M1H_fs : Real := -0.375;   // Активный ток статора, А (быстрое значение)
      su_W_M1H_fs : Real;   // Скорость, рад/с (быстрое значение)
      su_I_C_fs : Real;   // Действующий ток статора, A (быстрое значение)
      su_Id_C_fs : Real;   // Ток намагничивания статора, А (быстрое значение)
      su_Iq_C_fs : Real;   // Активный ток статора, А (быстрое значение)
      su_W_C_fs : Real;   // Скорость, рад/с (быстрое значение)
      su_I_S_fs : Real;   // Действующий ток статора, A (быстрое значение)
      su_Id_S_fs : Real;   // Ток намагничивания статора, А (быстрое значение)
      su_Iq_S_fs : Real := 59.75;   // Активный ток статора, А (быстрое значение)
      su_W_S_fs : Real;   // Скорость, рад/с (быстрое значение)
   END_VAR
BEGIN
END_DATA_BLOCK

DATA_BLOCK "AP"   // DB103
{ S7_Optimized_Access := 'FALSE' }
VERSION : 0.1
   VAR
      ap_QF_FanMD_Off : Bool;   // отключен автомат вентиляторов главных приводов
      ap_UZ_FanMD_On : Bool;   // преобразователь пуска вентиляторов главных приводов включен
      ap_QF_FanProp_Off : Bool;   // отключен автомат вентиляторов двигателей хода
      ap_UZ_FanProp_On : Bool;   // преобразователь пуска вентиляторов двигателей хода включен
      ap_QF_KB_On : Bool;   // автомат преобразователя кабельного барабана включен
      ap_QF_ODK_On : Bool;   // автомат преобразователя открывания днища ковша включен
      ap_PS_110v_On : Bool;   // питание источника 110В включено
      ap_CtrlC_110v_On : Bool;   // питание цепей управления 110В включено
      ap_Gudok : Bool;   // пневмосигнал включен
      ap_ODK : Bool;   // управление УДК
      ap_Vent_Prop_On : Bool;   // вентиляция привода хода включена
      ap_Vent_MD_On : Bool;   // вентиляция главных приводов включена
      ap_QF_FVU12_On : Bool;   // общий автомат ФВУ включен
      ap_FVU12_On : Bool;   // ФВУ включены
      ap_QF_FVU1_On : Bool;   // автомат ФВУ1 включен
      ap_QF_FVU2_On : Bool;   // автомат ФВУ2 включен
      ap_QF_Fan_Kuzov : Bool;   // автомат вентилятора кузова включен
      ap_Vent_Kuzov : Bool;   // вентиляция кузова включена
      ap_FVU1_FVU2_On : Bool;   // ФВУ1 или(и) ФВУ2 включен
      ap_QF_Lubr : Bool;   // общий автомат смазки редукторов поворота включен(0)
      ap_Lubr_On : Bool;   // смазка редукторов поворота включена
      ap_QF_Heat : Bool;   // общий автомат нагревателей смазки редукторов поворота включен
      ap_Heat_M1S : Bool;   // нагреватели ЕК1-ЕК6 включены
      ap_Heat_M2S : Bool;   // нагреватели ЕК7-ЕК12 включены
      ap_Heat_M3S : Bool;   // нагреватели ЕК13-ЕК18 включены
      ap_Heat_M4S : Bool;   // нагреватели ЕК19-ЕК23 включены
      ap_QF_Komr : Bool;   // компрессорная установка включена
      ap_QF_ACSS380V : Bool;   // станция густой смазки включена
      ap_QF_Vvod380 : Bool;   // вводной автоматический выключатель 380В включен
      ap_QF_TV3 : Bool;   // выключатель трансформатора TV3 включен
      ap_QF_TV2M : Bool;   // выключатель трансформатора TV2M включен
      ap_QF_Vent_SHGP : Bool;   // выключатель вентиляции ШГП включен
      ap_QF_Light : Bool;   // выключатель прожекторного освещения включен
      ap_QF_CtrlC24V : Bool;   // выключатель цепей управления -24В включен
      ap_QF_YAVV220V : Bool;   // выключатель цепей управления ЯВВ(220В) включен
      ap_QF_Charge_ZPT : Bool;   // выключатель цепей заряда конденсаторов включен
      ap_QF_BKTT220V : Bool;   // выключатель блока контроля температуры(220В) включен
      ap_QF_IS220V : Bool;   // выключатель ИС (220В) включен
      ap_QF_ACSS220V : Bool;   // выключатель обогрева шкафа густой смазки включен
      ap_KM_TV3 : Bool;   // трансформатор освещения TV3 включен
      ap_KM_Light : Bool;   // прожекторное освещение включен
      ap_KM_Heat_H : Bool;   // Контактор обогревателей масла редуктора подъЁма
      ap_QF_Heat_H : Bool;   // Автомат обогревателей масла редуктора подъЁма
   END_VAR
BEGIN
END_DATA_BLOCK

DATA_BLOCK "BD"   // DB120
{ S7_Optimized_Access := 'FALSE' }
VERSION : 0.1
   VAR
      n_Brig : Int;   // Номер бригады
      wt_H_Hour : DInt := DINT#0;   // Часы работы механизма подъёма
      wt_H_Minut : Int;   // Минуты работы механизма подъёма
      wt_H_Second : Int;   // Секунды работы механизма подъёма
      wt_C_Hour : DInt := DINT#0;   // Часы работы механизма напора
      wt_C_Minut : Int;   // Минуты работы механизма напора
      wt_C_Second : Int;   // Секунды работы механизма напора
      wt_S_Hour : DInt := DINT#0;   // Часы работы механизма поворота
      wt_S_Minut : Int;   // Минуты работы механизма поворота
      wt_S_Second : Int;   // Секунды работы механизма поворота
      wt_P_Hour : DInt := DINT#0;   // Часы работы механизма хода
      wt_P_Minut : Int;   // Минуты работы механизма хода
      wt_P_Second : Int;   // Секунды работы механизма хода
      wt_Exc_Hour : DInt := DINT#0;   // Время основной работы (Час)
      wt_Exc_Min : Int;   // Время основной работы (Минут)
      wt_Exc_Sec : Int;   // Время основной работы (Секунд)
      odo_Prop_all : Real;   // Общий пробег за время эксплуатации
      Spare_I_1 : Int;   // Резерв
      Spare_I_2 : Int;   // Резерв
      wt_Prop_Hour : DInt := DINT#0;   // Время хода (Час)
      wt_Prop_Min : Int;   // Время хода (Минут)
      wt_Prop_Sec : Int;   // Время хода (Секунд)
      wt_Idle_Hour : DInt := DINT#0;   // Время простоя (Час)
      wt_Idle_Min : Int;   // Время простоя (Минут)
      wt_Idle_Sec : Int;   // Время простоя (Секунд)
      wt_UG_Hour : DInt := DINT#0;   // Время работы при косом стоянии (Час)
      wt_UG_Min : Int;   // Время работы при косом стоянии (Минут)
      wt_UG_Sec : Int;   // Время работы при косом стоянии (Секунд)
      Mas_Basket : Real;   // Масса грунта в ковше (кг)
      Mas_TS_cr : Real;   // Масса грунта в ТС текущая (кг)
      Mas_TS_lst : Real;   // Масса грунта в последнем ТС (кг)
      Mas_TS_all : Real;   // Масса грунта общая (кг)
      AE1_st : Real;   // Активная потреблённая энергия в начале смены
      AE2_st : Real;   // Активная отданная энергия в начале смены
      RE1_st : Real;   // Реактивная потреблённая энергия в начале смены
      RE2_st : Real;   // Реактивная отданная энергия в начале смены
      AE1_cr : Real;   // Активная потреблённая энергия за смену
      AE2_cr : Real;   // Активная отданная энергия за смену
      RE1_cr : Real;   // Реактивная потреблённая энергия за смену
      RE2_cr : Real;   // Реактивная отданная энергия за смену
      AE1_all : Real;   // Активная потреблённая энергия общая
      AE2_all : Real;   // Активная отданная энергия общая
      RE1_all : Real;   // Реактивная потреблённая энергия общая
      RE2_all : Real;   // Реактивная отданная энергия общая
      tm_Reg_H : Int;   // Время регистрации бригады (час)
      tm_Reg_M : Int;   // Время регистрации бригады (мин)
      n_TS : Int;   // Количество погруженных ТС
      TS_Num : Int;   // Грузоподъёмность текущего ТС
      TS_1 : Int;   // Грузоподъёмность трансп.ср-ва 1
      TS_2 : Int;   // Грузоподъёмность трансп.ср-ва 2
      TS_3 : Int;   // Грузоподъёмность трансп.ср-ва 3
      TS_4 : Int;   // Грузоподъёмность трансп.ср-ва 4
      sm_Duration : Int;   // Продолжительность смены
      sm_Hour : Int;   // Начало первой смены. Час.
      sm_Min : Int;   // Начало первой смены. Мин.
      Shft_Reg : Bool;   // Флаг регистрации бригады
      fl_Pogr_On : Bool;   // Флаг погрузки
      Spare_160_2 : Bool;   // Резерв
      Spare_160_3 : Bool;   // Резерв
      Spare_160_4 : Bool;   // Резерв
      Spare_160_5 : Bool;   // Резерв
      Spare_160_6 : Bool;   // Резерв
      Spare_160_7 : Bool;   // Резерв
      tm_Reg_Mnt : Int;   // Время регистрации бригады (месяц)
      tm_Reg_Day : Int;   // Время регистрации бригады (год)
      kVAh_Total : DInt := DINT#0;   // Общая полная мощность
      Frequency : Real;   // Частота сети
      U_12 : Int;   // Напряжение между фазами 1 и 2
      U_23 : Int;   // Напряжение между фазами 2 и 3
      U_31 : Int;   // Напряжение между фазами 3 и 1
      PASS : Word;   // Эти три заглушки тут нужны чтобы адреса не съехали
      PASS1 : Word;   // Эти три заглушки тут нужны чтобы адреса не съехали
      PASS2 : Word;   // Эти три заглушки тут нужны чтобы адреса не съехали
      I_1 : Real;   // Ток фазы 1
      I_2 : Real;   // Ток фазы 2
      I_3 : Real;   // Ток фазы 3
      PF : Real;   // Сдвиг фаз
      Count_BTL_ErrPoint_2 : Int;   // Количество забросов за вторую точку
   END_VAR
BEGIN
END_DATA_BLOCK

DATA_BLOCK "Work"   // DB121
TITLE = Данные для работы
{ S7_Optimized_Access := 'FALSE' }
VERSION : 0.1
   VAR
      on_SU : Bool;   // Система управления в работе
      pH_On : Bool;   // Привод подьёма включен
      pS_On : Bool;   // Привод поворота включен
      pC_On : Bool;   // Привод напора включен
      pP_On : Bool;   // Привод хода включен
      p_On : Bool;   // Главные приводы включены
      ACSS_On : Bool;   // АЦСС в работе
      HMI_On : Bool;   // HMI в работе
      Auto_Park : Bool;   // Команда на автоматическую парковку компьютера
      Ack_Alrm : Bool;   // Квитирование алармов
      T_Set_on : Bool;   // Команда на установку времени
      fl_Reset_LH : Bool;   // Флаг сброса длины каната подъёма
      fl_Reset_LC : Bool;   // Флаг сброса длины рукояти
      on_Auto_Def : Bool;   // Включение / отключение автозащит
      Reset_flt_SU : Bool;   // Сброс ошибок системы управления
      LK_ON : Bool;   // Вывод левой камеры
      cnt_Sec : Int;   // Счётчик секунд
      ABS_U : Int;   // Абсолютный угол поворота
      Spare_w6 : Word;   // Уставка паузы P1
      ug_Prod_Mx : Real;   // Угол наклона экскаватора продольная плоскость предыдущий
      ug_Popr_Mx : Real;   // Угол наклона экскаватора поперечная плоскость предыдущий
      ug_Prod_Mn : Real;   // Разность между тек. и пред. уголаами в продольной плоскости
      ug_Popr_Mn : Real;   // Разность между тек. и пред. уголаами в поперечной плоскости
      ug_Prod_MAX : Real;   // Разность между тек. и пред. уголаами в продольной плоскости макс.
      ug_Popr_MAX : Real;   // Разность между тек. и пред. уголаами в поперечной плоскости макс.
      ABS_H : Real;   // Абсолютная скорость подъёма
      Spare_I36 : Int;   // Счётчик лайфбитов АЦСС
      Spare_I38 : Int;   // Предыдущий лайфбит АЦСС
      HMI_LB : Int;   // Лайфбит HMI
      HMI_LB_Cnt : Int;   // Счётчик лайфбитов HMI
      HMI_LB_Pred : Int;   // Предыдущий лайфбит HMI
      smf_ACSS : Int;   // Суммарный фолт системы смазки
      smf_Tmpr : Int;   // Суммарный фолт температур
      Act_Time_Year : Int;   // Текущая дата/время - Год
      Act_Time_Month : Int;   // Текущая дата/время - Месяц
      Act_Time_Day : Int;   // Текущая дата/время - День
      Act_Time_Hour : Int;   // Текущая дата/время - Час
      Act_Time_Min : Int;   // Текущая дата/время - Минуты
      Act_Time_Sec : Int;   // Текущая дата/время - Секунды
      smf_AP : Int;   // Суммарный фолт вспомогательных приводов
      smf_GP : Int;   // Суммарный фолт главных приводов
      fl_WC_Start : Bool;   // Флаг начала рабочего цикла
      Spare_66_1 : Bool;   // Резерв
      Spare_66_2 : Bool;   // Резерв
      Reg_Lim_BN : Bool;   // Режим ограничения по боковым нагрузкам
      fl_Blok_BN : Bool;   // Флаг блокировки защиты от боковых нагрузок
      fl_Kach : Bool;   // Флаг измерения качания
      fl_S_Final : Bool;   // Флаг завершения смены
      Spare_66_7 : Bool;   // Резерв
      fl_WC_Idle : Bool;   // Флаг простоя
      fl_WC_Drag : Bool;   // Флаг черпания
      fl_WC_S_Rz : Bool;   // Флаг поворота разгрузку
      fl_WC_Rz : Bool;   // Флаг разгрузи
      fl_WC_S_Zb : Bool;   // Флаг поворота в забой
      fl_WC_Prop : Bool;   // Флаг хода
      fl_WC_Wait : Bool;   // Флаг ожидания транспорта
      Spare_67_7 : Bool;   // Резерв
      Spare_W68 : Word;   // Резерв
      lim_VH : Byte;   // Ограничение скорости подъёма
      lim_VS : Byte;   // Ограничение скорости поворота
      lim_VC : Byte;   // Ограничение скорости напора
      lim_IsH : Byte;   // Ограничение стопорного тока подъёма
      lim_IsS : Byte;   // Ограничение стопорного тока поворота
      lim_IsC : Byte;   // Ограничение стопорного тока напора
      ug_Pov_Tk : Int;   // Угол поворота платформы экскаватора текущий
      cmd_SU : Byte;   // Команда системе управления
      cnt_Zub : Int;   // Счётчик зубъев
      fl_Entg_Res : Bool;   // Флаг сброса счётчика
      Win_Protect : Bool;   // Флаг работы в зимнее время
      Shft_f_Reg : Bool;   // Флаг первой регистрации бригады
      fl_Excs : Bool;   // Флаг экскавации
      fl_Prop : Bool;   // Флаг перемещения
      fl_Idle : Bool;   // Флаг простоя
      Camera_ON : Bool;   // Включение камеры
      Camera_FIN : Bool;   // Отключение камеры
      fl_Second : Bool;   // Фронт секунд
      Reg_Lim_Turn : Bool;   // Режим ограничений от недопустимого разворота
      Reset_Enrg : Bool;   // Сброс счётчика
      fl_KS : Bool;   // Флаг работы при косом стоянии
      Winter_Pr_Removing : Bool;   // Процесс снятия зимних защит запущен
      ACSS_Starting_Now : Bool;   // Выполняется запуск системы смазки (0-нет; 1-да)
      ACSS_SumBypass : Bool;   // Суммарный байпасс питателей системы смазки
      RB_HMI : Bool;   // Эмулятор правой кнопки командоаппарата с HMI
      Camera_Reg : Int;   // Режим работы камеры
      smf_Komp : Int;   // Суммарный фолт компрессора
      ABS_Sw : Real;   // Абсолютная скорость поворота
      Reg_WC : Int;   // Режим рабочего цикла (1-черпание,2-пов.на разгр,3-разгр,4-поворот в заб.)
      ug_Povorota : Int;   // Угол поворота платформы экскаватора
      Prc_TS : Int;   // Процент заполнения самосвала
      dp_ET_2 : Bool;   // Флаг работы станции ET200 в шкафу АИС2
      dp_ET_3 : Bool;   // Флаг работы станции ET200 в шкафу АИС3
      dp_ET_4 : Bool;   // Флаг работы станции ET200 в шкафу АИС4
      dp_ACSS : Bool;   // Флаг работы контроллера густой смазки
      dp_CAN_AP : Bool;   // Флаг работы шлюза CAN-DP вспом. приводов
      dp_CAN_GP : Bool;   // Флаг работы шлюза CAN-DP гл. приводов
      dp_GNAMG : Bool;   // Флаг работы инклинометра
      dp_KOMPR : Bool;   // Флаг работы компрессора
      fl_Wint_Pr : Bool;   // Флаг защиты МК при работе зимой
      fl_Win_Pr_St_Res : Bool;   // Флаг старта процедуры сброса
      Reg_Lim_UG : Bool;   // Режим ограничения по углу стояния
      Reg_Lim_ZS : Bool;   // Режим ограничения от заброса стрелы
      Reg_Lim_Winter : Bool;   // Режим ограничения зимой
      Reg_Lim_HMI : Bool;   // Режим ограничения с HMI
      bl_Rdy : Bool;   // Флаг готовности БУП к обработке сообщений
      bl_A_Rdy : Bool;   // Флаг готовности БУАВ к обработке сообщений
      DT_Wint_Res : Date_And_Time;   // Дата и время отключения защит в зимнее время
      lb_PLC : Int;   // Лайфбит PLC
      smf_ACSS_A1 : Int;   // Суммарный фолт станции A1 системы смазки
      smf_ACSS_A2 : Int;   // Суммарный фолт станции A2 системы смазки
      smf_ACSS_H1 : Int;   // Суммарный фолт станции H1 системы смазки
      tm_WP_Reset : DInt := DINT#0;   // Время до снятия зимних защит mc
      Offset : Int;   // Сдвиг в блоке данных старых алармов
      lim_VH_HMI : Byte;   // Ограничение скорости подъёма с HMI
      lim_VS_HMI : Byte;   // Ограничение скорости поворота с HMI
      lim_VC_HMI : Byte;   // Ограничение скорости напора с HMI
      lim_IsH_HMI : Byte;   // Ограничение стопорного тока подъёма с HMI
      lim_IsS_HMI : Byte;   // Ограничение стопорного тока поворота с HMI
      lim_IsC_HMI : Byte;   // Ограничение стопорного тока напора с HMI
      n_BUP_cr : Int;   // Текущий номер БУП
      n_BUP_pr : Int;   // Предыдущий номер БУП
      cnt_BUP : Int;   // Счётчик БУП
      n_BUP : Array[1..15] of Int;   // Массив номеров блоков
      t_BUP : Array[1..15] of Int;   // Массив типов блоков
      SU_LB : Int;   // Лайфбит СУ
      SU_LB_Cnt : Int;   // Счётчик лайфбитов СУ
      SU_LB_Pred : Int;   // Предыдущий лайфбит СУ
      QwrSATEC : DWord;   // Формируемое двойное слово запроса, отправляемое в счётчик электроэнергии
      PASS_SATEC : DWord := DWORD#16#0101_0E14;   // Заготовка для посылки: byte0(0001 0100)byte1(0000 1110)ID-0x0101
      Control_Run_FC114 : Int;   // Здесь лежит байт, управляющий чтением показаний с SADEC
      su_LH_prev : Real;   // Предыдущая (50Гц) длина подъемного каната м
      su_LC_prev : Real;   // Предыдущая (50Гц) длина выдвижения рукояти м
      V_prop_left : Real;   // Скорость движения левой гусеницы
      V_prop_right : Real;   // Скорость движения правой гусеницы
      su_W_M1P_Pred : Real;   // Скорость двигателя хода M1P в предыдущем скане
      su_W_M2P_Pred : Real;   // Скорость двигателя хода M2P в предыдущем скане
      W_pP_Pred : Real;   // Cредняя скорость привода хода в предыдущем скане
      W_pP_Cr : Real;   // Cредняя скорость привода хода в текущем скане
      ABS_W_pP_Pred : Real;   // Абсолютное значение средней скорости привода хода в предыдущем скане
      ABS_W_pP_Cr : Real;   // Абсолютное значение средней скорости привода хода в текущем скане
      odo_Prop_cr : Real;   // Пробег за один шаг интегрирования
      lim_VP_M1P : Byte;   // Ограничение скорости левой гусеницы
      lim_VP_M2p : Byte;   // Ограничение скорости правой гусеницы
   END_VAR
BEGIN
END_DATA_BLOCK

DATA_BLOCK "DB_OSC"   // DB505
{ S7_Optimized_Access := 'FALSE' }
VERSION : 0.1
   VAR
      Act : Int;   // Флаг работы осцилографа
      Ready : Int;   // Флаг готовности массивов к передаче
      Cnt : Int;   // Счётчик параметров
      Ramp : Int;   // Пила
      Max_Addr : DInt := DINT#0;   // Максимальный адрес текущего массива
      cr_Addr_1 : DInt := DINT#0;   // Текущий адрес массива канала 1
      cr_Addr_2 : DInt := DINT#0;   // Текущий адрес массива канала 2
      cr_Addr_3 : DInt := DINT#0;   // Текущий адрес массива канала 3
      cr_Addr_4 : DInt := DINT#0;   // Текущий адрес массива канала 4
      cr_Addr_5 : DInt := DINT#0;   // Текущий адрес массива канала 5
      cr_Addr_6 : DInt := DINT#0;   // Текущий адрес массива канала 6
      cr_Addr_7 : DInt := DINT#0;   // Текущий адрес массива канала 7
      cr_Addr_8 : DInt := DINT#0;   // Текущий адрес массива канала 8
      cr_Addr_9 : DInt := DINT#0;   // Текущий адрес массива канала 9
      cr_Addr_10 : DInt := DINT#0;   // Текущий адрес массива канала 10
      cr_Addr_Rmp : DInt := DINT#32448;   // Текущий адрес пилы
      ar_Ch_01 : Array[1..200] of Int;   // Массив значений канала 1
      ar_Ch_02 : Array[1..200] of Int;   // Массив значений канала 2
      ar_Ch_03 : Array[1..200] of Int;   // Массив значений канала 3
      ar_Ch_04 : Array[1..200] of Int;   // Массив значений канала 4
      ar_Ch_05 : Array[1..200] of Int;   // Массив значений канала 5
      ar_Ch_06 : Array[1..200] of Int;   // Массив значений канала 6
      ar_Ch_07 : Array[1..200] of Int;   // Массив значений канала 7
      ar_Ch_08 : Array[1..200] of Int;   // Массив значений канала 8
      ar_Ch_09 : Array[1..200] of Int;   // Массив значений канала 9
      ar_Ch_10 : Array[1..200] of Int;   // Массив значений канала 10
      ar_Ramp : Array[1..200] of Int;   // Массив значений с пилой
      Ch_1 : Int;   // Текущее значение канала 1
      Ch_2 : Int;   // Текущее значение канала 2
      Ch_3 : Int;   // Текущее значение канала 3
      Ch_4 : Int;   // Текущее значение канала 4
      Ch_5 : Int;   // Текущее значение канала 5
      Ch_6 : Int;   // Текущее значение канала 6
      Ch_7 : Int;   // Текущее значение канала 7
      Ch_8 : Int;   // Текущее значение канала 8
      Ch_9 : Int;   // Текущее значение канала 9
      Ch_10 : Int;   // Текущее значение канала 10
   END_VAR
BEGIN
   ar_Ch_01[17] := 276;
END_DATA_BLOCK

FUNCTION "OSC" : Void   // FC500, STL
{ S7_Optimized_Access := 'FALSE' }
VERSION : 0.1
   VAR_TEMP
      CH_10 : Int;
      CH_09 : Int;
      CH_08 : Int;
      CH_07 : Int;
      CH_06 : Int;
      CH_05 : Int;
      CH_04 : Int;
      CH_03 : Int;
      CH_02 : Int;
      CH_01 : Int;
      TMP_DI : DInt;
      For_SIN : Int;   // тест можно удалить
      For_Ramp : Int;   // тест можно удалить
      For_Square : Int;   // тест можно удалить
      For_TriangleUp : Int;   // тест можно удалить
   END_VAR
BEGIN

REGION Network 1: признак прироста треугольника вверх

   //      CALL  "OSC_BS_GP"
   //         Ch_01 :=#CH_01
   //         Ch_02 :=#CH_02
   //         Ch_03 :=#CH_03
   //         Ch_04 :=#CH_04
   //         Ch_05 :=#CH_05
   //         Ch_06 :=#CH_06
   //         Ch_07 :=#CH_07
   //         Ch_08 :=#CH_08
   //         Ch_09 :=#CH_09
   //         Ch_10 :=#CH_10

   //      CALL  "Bl_Spr_OE"
   //       Ch_01:=#CH_01
   //       Ch_02:=#CH_02
   //       Ch_03:=#CH_03
   //       Ch_04:=#CH_04
   //       Ch_05:=#CH_05
   //       Ch_06:=#CH_06
   //       Ch_07:=#CH_07
   //       Ch_08:=#CH_08
   //       Ch_09:=#CH_09
   //       Ch_10:=#CH_10

   //      CALL  FC   514
   //       Ch_01:=#CH_01
   //       Ch_02:=#CH_02
   //       Ch_03:=#CH_03
   //       Ch_04:=#CH_04
   //       Ch_05:=#CH_05
   //       Ch_06:=#CH_06
   //       Ch_07:=#CH_07
   //       Ch_08:=#CH_08
   //       Ch_09:=#CH_09
   //       Ch_10:=#CH_10

   // треугольник верхний

         AN    "Temp".If_Up;
         JNB   _009;

         L     "Temp".TriangleUp;
         L     20.0;
         -R;
         T     "Temp".TriangleUp;

